LIN {X 0,Y 446.601,Z 250.355,A -85,B 0,C 180,E1 -8646.329,E2 -8646.329} C_VEL
LIN {X 0,Y 446.522,Z 250.36,A -85,B 0,C 180,E1 -8649.06,E2 -8649.06} C_VEL
LIN {X 0,Y 446.522,Z 250.36,A -85,B 0,C 180,E1 -8652.734,E2 -8652.734} C_VEL
LIN {X 0,Y 446.451,Z 250.372,A -85,B 0,C 180,E1 -8656.211,E2 -8656.211} C_VEL
LIN {X 0,Y 446.47,Z 250.369,A -85,B 0,C 180,E1 -8659.307,E2 -8659.307} C_VEL
LIN {X 0,Y 446.419,Z 250.374,A -85,B 0,C 180,E1 -8662.204,E2 -8662.204} C_VEL
LIN {X 0,Y 446.426,Z 250.375,A -85,B 0,C 180,E1 -8665.158,E2 -8665.158} C_VEL
LIN {X 0,Y 446.422,Z 250.373,A -85,B 0,C 180,E1 -8668.187,E2 -8668.187} C_VEL
LIN {X 0,Y 446.415,Z 250.38,A -85,B 0,C 180,E1 -8671.304,E2 -8671.304} C_VEL
LIN {X 0,Y 446.428,Z 250.375,A -85,B 0,C 180,E1 -8674.527,E2 -8674.527} C_VEL
LIN {X 0,Y 446.414,Z 250.379,A -85,B 0,C 180,E1 -8678.08,E2 -8678.08} C_VEL
LIN {X 0,Y 446.421,Z 250.437,A -85,B 0,C 180,E1 -8681.396,E2 -8681.396} C_VEL
LIN {X 0,Y 447.055,Z 254.418,A -85,B 0,C 180,E1 -8685.03,E2 -8685.03} C_VEL
LIN {X 0,Y 447.395,Z 257.531,A -85,B 0,C 180,E1 -8687.592,E2 -8687.592} C_VEL
LIN {X 0,Y 447.38,Z 261.124,A -85,B 0,C 180,E1 -8690.336,E2 -8690.336} C_VEL
LIN {X 0,Y 447.027,Z 265.384,A -85,B 0,C 180,E1 -8693.315,E2 -8693.315} C_VEL
LIN {X 0,Y 446.739,Z 270.172,A -85,B 0,C 180,E1 -8696.494,E2 -8696.494} C_VEL
LIN {X 0,Y 446.406,Z 275.403,A -85,B 0,C 180,E1 -8699.749,E2 -8699.749} C_VEL
LIN {X 0,Y 446.193,Z 280.555,A -85,B 0,C 180,E1 -8702.821,E2 -8702.821} C_VEL
LIN {X 0,Y 445.943,Z 285.793,A -85,B 0,C 180,E1 -8705.811,E2 -8705.811} C_VEL
LIN {X 0,Y 445.831,Z 291.111,A -85,B 0,C 180,E1 -8708.742,E2 -8708.742} C_VEL
LIN {X 0,Y 445.64,Z 296.456,A -85,B 0,C 180,E1 -8711.615,E2 -8711.615} C_VEL
LIN {X 0,Y 445.564,Z 300.748,A -85,B 0,C 180,E1 -8713.868,E2 -8713.868} C_VEL
LIN {X 0,Y 447.507,Z 311.304,A -85,B 0,C 180,E1 -8714.232,E2 -8714.232} C_VEL
LIN {X 0,Y 449.155,Z 321.497,A -85,B 0,C 180,E1 -8714.69,E2 -8714.69} C_VEL
LIN {X 0,Y 449.183,Z 328.569,A -85,B 0,C 180,E1 -8715.039,E2 -8715.039} C_VEL
LIN {X 0,Y 448.687,Z 338.087,A -85,B 0,C 180,E1 -8715.602,E2 -8715.602} C_VEL
LIN {X 0,Y 448.174,Z 347.367,A -85,B 0,C 180,E1 -8716.28,E2 -8716.28} C_VEL
LIN {X 0,Y 447.792,Z 355.767,A -85,B 0,C 180,E1 -8717.021,E2 -8717.021} C_VEL
LIN {X 0,Y 447.286,Z 364.854,A -85,B 0,C 180,E1 -8717.984,E2 -8717.984} C_VEL
LIN {X 0,Y 446.839,Z 372.076,A -85,B 0,C 180,E1 -8718.891,E2 -8718.891} C_VEL
LIN {X 0,Y 446.495,Z 378.281,A -85,B 0,C 180,E1 -8719.801,E2 -8719.801} C_VEL
LIN {X 0,Y 446.129,Z 384.821,A -85,B 0,C 180,E1 -8720.936,E2 -8720.936} C_VEL
LIN {X 0,Y 445.891,Z 389.324,A -85,B 0,C 180,E1 -8721.845,E2 -8721.845} C_VEL
LIN {X 0,Y 445.666,Z 394.973,A -85,B 0,C 180,E1 -8723.253,E2 -8723.253} C_VEL
LIN {X 0,Y 445.537,Z 399.142,A -85,B 0,C 180,E1 -8724.569,E2 -8724.569} C_VEL
LIN {X 0,Y 445.431,Z 401.507,A -85,B 0,C 180,E1 -8725.475,E2 -8725.475} C_VEL
LIN {X 0,Y 445.391,Z 403.304,A -85,B 0,C 180,E1 -8726.381,E2 -8726.381} C_VEL
LIN {X 0,Y 445.357,Z 405.747,A -85,B 0,C 180,E1 -8728.191,E2 -8728.191} C_VEL
LIN {X 0,Y 445.32,Z 406.334,A -85,B 0,C 180,E1 -8729.096,E2 -8729.096} C_VEL
LIN {X 0,Y 445.32,Z 406.334,A -85,B 0,C 180,E1 -8730.904,E2 -8730.904} C_VEL
LIN {X 0,Y 445.357,Z 405.747,A -85,B 0,C 180,E1 -8731.809,E2 -8731.809} C_VEL
LIN {X 0,Y 445.391,Z 403.304,A -85,B 0,C 180,E1 -8733.619,E2 -8733.619} C_VEL
LIN {X 0,Y 445.503,Z 400.359,A -85,B 0,C 180,E1 -8734.977,E2 -8734.977} C_VEL
LIN {X 0,Y 445.59,Z 396.371,A -85,B 0,C 180,E1 -8736.339,E2 -8736.339} C_VEL
LIN {X 0,Y 445.768,Z 391.24,A -85,B 0,C 180,E1 -8737.701,E2 -8737.701} C_VEL
LIN {X 0,Y 446.082,Z 385.978,A -85,B 0,C 180,E1 -8738.836,E2 -8738.836} C_VEL
LIN {X 0,Y 446.427,Z 379.658,A -85,B 0,C 180,E1 -8739.972,E2 -8739.972} C_VEL
LIN {X 0,Y 446.724,Z 373.703,A -85,B 0,C 180,E1 -8740.882,E2 -8740.882} C_VEL
LIN {X 0,Y 447.158,Z 366.773,A -85,B 0,C 180,E1 -8741.79,E2 -8741.79} C_VEL
LIN {X 0,Y 447.622,Z 358.589,A -85,B 0,C 180,E1 -8742.698,E2 -8742.698} C_VEL
LIN {X 0,Y 448.02,Z 350.084,A -85,B 0,C 180,E1 -8743.493,E2 -8743.493} C_VEL
LIN {X 0,Y 448.505,Z 341.352,A -85,B 0,C 180,E1 -8744.172,E2 -8744.172} C_VEL
LIN {X 0,Y 449,Z 331.59,A -85,B 0,C 180,E1 -8744.793,E2 -8744.793} C_VEL
LIN {X 0,Y 449.343,Z 322.793,A -85,B 0,C 180,E1 -8745.245,E2 -8745.245} C_VEL
LIN {X 0,Y 447.629,Z 311.904,A -85,B 0,C 180,E1 -8745.743,E2 -8745.743} C_VEL
LIN {X 0,Y 445.696,Z 301.798,A -85,B 0,C 180,E1 -8746.101,E2 -8746.101} C_VEL
LIN {X 0,Y 445.565,Z 300.694,A -85,B 0,C 180,E1 -8746.16,E2 -8746.16} C_VEL
LIN {X 0,Y 445.696,Z 294.655,A -85,B 0,C 180,E1 -8749.338,E2 -8749.338} C_VEL
LIN {X 0,Y 445.858,Z 289.313,A -85,B 0,C 180,E1 -8752.229,E2 -8752.229} C_VEL
LIN {X 0,Y 446.154,Z 282.386,A -85,B 0,C 180,E1 -8756.113,E2 -8756.113} C_VEL
LIN {X 0,Y 446.347,Z 277.096,A -85,B 0,C 180,E1 -8759.216,E2 -8759.216} C_VEL
LIN {X 0,Y 446.615,Z 271.991,A -85,B 0,C 180,E1 -8762.345,E2 -8762.345} C_VEL
LIN {X 0,Y 446.91,Z 266.987,A -85,B 0,C 180,E1 -8765.58,E2 -8765.58} C_VEL
LIN {X 0,Y 447.299,Z 262.126,A -85,B 0,C 180,E1 -8768.937,E2 -8768.937} C_VEL
LIN {X 0,Y 447.437,Z 258.971,A -85,B 0,C 180,E1 -8771.276,E2 -8771.276} C_VEL
LIN {X 0,Y 447.266,Z 255.884,A -85,B 0,C 180,E1 -8773.739,E2 -8773.739} C_VEL
LIN {X 0,Y 446.779,Z 252.867,A -85,B 0,C 180,E1 -8776.351,E2 -8776.351} C_VEL
LIN {X 0,Y 446.421,Z 250.435,A -85,B 0,C 180,E1 -8778.604,E2 -8778.604} C_VEL
LIN {X 0,Y 446.412,Z 250.379,A -85,B 0,C 180,E1 -8781.92,E2 -8781.92} C_VEL
LIN {X 0,Y 446.428,Z 250.374,A -85,B 0,C 180,E1 -8785.473,E2 -8785.473} C_VEL
LIN {X 0,Y 446.415,Z 250.38,A -85,B 0,C 180,E1 -8788.696,E2 -8788.696} C_VEL
LIN {X 0,Y 446.43,Z 250.372,A -85,B 0,C 180,E1 -8791.833,E2 -8791.833} C_VEL
LIN {X 0,Y 446.426,Z 250.375,A -85,B 0,C 180,E1 -8794.842,E2 -8794.842} C_VEL
LIN {X 0,Y 446.451,Z 250.375,A -85,B 0,C 180,E1 -8798.242,E2 -8798.242} C_VEL
LIN {X 0,Y 446.44,Z 250.372,A -85,B 0,C 180,E1 -8801.644,E2 -8801.644} C_VEL
LIN {X 0,Y 446.459,Z 250.371,A -85,B 0,C 180,E1 -8804.474,E2 -8804.474} C_VEL
LIN {X 0,Y 446.516,Z 250.362,A -85,B 0,C 180,E1 -8807.379,E2 -8807.379} C_VEL
LIN {X 0,Y 446.522,Z 250.36,A -85,B 0,C 180,E1 -8810.94,E2 -8810.94} C_VEL
LIN {X 0,Y 446.601,Z 250.355,A -85,B 0,C 180,E1 -8813.671,E2 -8813.671} C_VEL
LIN {X 0,Y 446.646,Z 250.347,A -85,B 0,C 180,E1 -8817.289,E2 -8817.289} C_VEL
LIN {X 0,Y 446.709,Z 250.341,A -85,B 0,C 180,E1 -8819.995,E2 -8819.995} C_VEL
LIN {X 0,Y 446.669,Z 250.342,A -85,B 0,C 180,E1 -8822.7,E2 -8822.7} C_VEL
LIN {X 0,Y 446.614,Z 250.349,A -85,B 0,C 180,E1 -8826.318,E2 -8826.318} C_VEL
LIN {X 0,Y 446.516,Z 250.364,A -85,B 0,C 180,E1 -8829.05,E2 -8829.05} C_VEL
LIN {X 0,Y 446.504,Z 250.364,A -85,B 0,C 180,E1 -8832.724,E2 -8832.724} C_VEL
LIN {X 0,Y 446.467,Z 250.367,A -85,B 0,C 180,E1 -8836.453,E2 -8836.453} C_VEL
LIN {X 0,Y 446.444,Z 250.375,A -85,B 0,C 180,E1 -8839.298,E2 -8839.298} C_VEL
LIN {X 0,Y 446.391,Z 250.377,A -85,B 0,C 180,E1 -8842.194,E2 -8842.194} C_VEL
LIN {X 0,Y 446.417,Z 250.378,A -85,B 0,C 180,E1 -8845.147,E2 -8845.147} C_VEL
LIN {X 0,Y 446.453,Z 250.369,A -85,B 0,C 180,E1 -8848.173,E2 -8848.173} C_VEL
LIN {X 0,Y 446.383,Z 250.377,A -85,B 0,C 180,E1 -8851.769,E2 -8851.769} C_VEL
LIN {X 0,Y 446.393,Z 250.382,A -85,B 0,C 180,E1 -8854.517,E2 -8854.517} C_VEL
LIN {X 0,Y 446.372,Z 250.381,A -85,B 0,C 180,E1 -8858.073,E2 -8858.073} C_VEL
LIN {X 0,Y 446.393,Z 250.376,A -85,B 0,C 180,E1 -8861.385,E2 -8861.385} C_VEL
LIN {X 0,Y 446.411,Z 250.375,A -85,B 0,C 180,E1 -8864.892,E2 -8864.892} C_VEL
LIN {X 0,Y 446.403,Z 250.376,A -85,B 0,C 180,E1 -8867.715,E2 -8867.715} C_VEL
LIN {X 0,Y 446.423,Z 250.373,A -85,B 0,C 180,E1 -8870.972,E2 -8870.972} C_VEL
LIN {X 0,Y 446.367,Z 250.383,A -85,B 0,C 180,E1 -8874.37,E2 -8874.37} C_VEL
LIN {X 0,Y 446.373,Z 250.382,A -85,B 0,C 180,E1 -8877.635,E2 -8877.635} C_VEL
LIN {X 0,Y 446.411,Z 250.374,A -85,B 0,C 180,E1 -8880.789,E2 -8880.789} C_VEL
LIN {X 0,Y 446.418,Z 250.38,A -85,B 0,C 180,E1 -8883.845,E2 -8883.845} C_VEL
LIN {X 0,Y 446.387,Z 250.377,A -85,B 0,C 180,E1 -8886.821,E2 -8886.821} C_VEL
LIN {X 0,Y 446.397,Z 250.382,A -85,B 0,C 180,E1 -8889.735,E2 -8889.735} C_VEL
LIN {X 0,Y 446.408,Z 250.378,A -85,B 0,C 180,E1 -8892.595,E2 -8892.595} C_VEL
LIN {X 0,Y 446.423,Z 250.38,A -85,B 0,C 180,E1 -8895.411,E2 -8895.411} C_VEL
LIN {X 0,Y 446.482,Z 250.368,A -85,B 0,C 180,E1 -8898.192,E2 -8898.192} C_VEL
LIN {X 0,Y 446.54,Z 250.362,A -85,B 0,C 180,E1 -8901.857,E2 -8901.857} C_VEL
LIN {X 0,Y 446.591,Z 250.356,A -85,B 0,C 180,E1 -8904.582,E2 -8904.582} C_VEL
LIN {X 0,Y 446.56,Z 250.36,A -85,B 0,C 180,E1 -8906.966,E2 -8906.966} C_VEL
LIN {X 0,Y 446.041,Z 250.428,A -85,B 0,C 180,E1 -8907.719,E2 -8907.719} C_VEL
LIN {X 0,Y 443.252,Z 250.781,A -85,B 0,C 180,E1 -8908.943,E2 -8908.943} C_VEL
LIN {X 0,Y 440.785,Z 251.087,A -85,B 0,C 180,E1 -8909.93,E2 -8909.93} C_VEL
LIN {X 0,Y 439.691,Z 251.219,A -85,B 0,C 180,E1 -8910.693,E2 -8910.693} C_VEL
LIN {X 0,Y 439.588,Z 251.229,A -85,B 0,C 180,E1 -8910.952,E2 -8910.952} C_VEL
LIN {X 0,Y 439.599,Z 251.229,A -85,B 0,C 180,E1 -8912.749,E2 -8912.749} C_VEL
LIN {X 0,Y 439.567,Z 251.233,A -85,B 0,C 180,E1 -8916.426,E2 -8916.426} C_VEL
LIN {X 0,Y 439.452,Z 251.246,A -85,B 0,C 180,E1 -8919.202,E2 -8919.202} C_VEL
LIN {X 0,Y 439.44,Z 251.25,A -85,B 0,C 180,E1 -8922.728,E2 -8922.728} C_VEL
LIN {X 0,Y 439.397,Z 251.254,A -85,B 0,C 180,E1 -8926.357,E2 -8926.357} C_VEL
LIN {X 0,Y 439.373,Z 251.251,A -85,B 0,C 180,E1 -8929.627,E2 -8929.627} C_VEL
LIN {X 0,Y 439.325,Z 251.261,A -85,B 0,C 180,E1 -8932.577,E2 -8932.577} C_VEL
LIN {X 0,Y 439.355,Z 251.254,A -85,B 0,C 180,E1 -8935.587,E2 -8935.587} C_VEL
LIN {X 0,Y 439.367,Z 251.253,A -85,B 0,C 180,E1 -8938.676,E2 -8938.676} C_VEL
LIN {X 0,Y 439.328,Z 251.264,A -85,B 0,C 180,E1 -8942.037,E2 -8942.037} C_VEL
LIN {X 0,Y 439.341,Z 251.256,A -85,B 0,C 180,E1 -8945.345,E2 -8945.345} C_VEL
LIN {X 0,Y 439.347,Z 251.254,A -85,B 0,C 180,E1 -8948.598,E2 -8948.598} C_VEL
LIN {X 0,Y 439.355,Z 251.255,A -85,B 0,C 180,E1 -8951.264,E2 -8951.264} C_VEL
LIN {X 0,Y 439.363,Z 251.252,A -85,B 0,C 180,E1 -8954.733,E2 -8954.733} C_VEL
LIN {X 0,Y 439.367,Z 251.256,A -85,B 0,C 180,E1 -8957.803,E2 -8957.803} C_VEL
LIN {X 0,Y 439.347,Z 251.254,A -85,B 0,C 180,E1 -8960.229,E2 -8960.229} C_VEL
LIN {X 0,Y 439.336,Z 251.259,A -85,B 0,C 180,E1 -8963.718,E2 -8963.718} C_VEL
LIN {X 0,Y 439.337,Z 251.26,A -85,B 0,C 180,E1 -8967.06,E2 -8967.06} C_VEL
LIN {X 0,Y 439.348,Z 251.254,A -85,B 0,C 180,E1 -8970.28,E2 -8970.28} C_VEL
LIN {X 0,Y 439.398,Z 251.251,A -85,B 0,C 180,E1 -8973.402,E2 -8973.402} C_VEL
LIN {X 0,Y 439.357,Z 251.254,A -85,B 0,C 180,E1 -8976.435,E2 -8976.435} C_VEL
LIN {X 0,Y 439.362,Z 251.254,A -85,B 0,C 180,E1 -8979.403,E2 -8979.403} C_VEL
LIN {X 0,Y 439.381,Z 251.251,A -85,B 0,C 180,E1 -8982.314,E2 -8982.314} C_VEL
LIN {X 0,Y 439.423,Z 251.247,A -85,B 0,C 180,E1 -8985.18,E2 -8985.18} C_VEL
LIN {X 0,Y 439.466,Z 251.24,A -85,B 0,C 180,E1 -8988.007,E2 -8988.007} C_VEL
LIN {X 0,Y 439.489,Z 251.236,A -85,B 0,C 180,E1 -8991.731,E2 -8991.731} C_VEL
LIN {X 0,Y 439.596,Z 251.23,A -85,B 0,C 180,E1 -8994.501,E2 -8994.501} C_VEL
LIN {X 0,Y 439.623,Z 251.225,A -85,B 0,C 180,E1 -8998.173,E2 -8998.173} C_VEL
LIN {X 0,Y 439.577,Z 251.226,A -85,B 0,C 180,E1 -9000.921,E2 -9000.921} C_VEL
LIN {X 0,Y 439.597,Z 251.224,A -85,B 0,C 180,E1 -9002.754,E2 -9002.754} C_VEL
LIN {X 0,Y 439.554,Z 251.232,A -85,B 0,C 180,E1 -9006.431,E2 -9006.431} C_VEL
LIN {X 0,Y 439.487,Z 251.237,A -85,B 0,C 180,E1 -9009.207,E2 -9009.207} C_VEL
LIN {X 0,Y 439.465,Z 251.239,A -85,B 0,C 180,E1 -9012.942,E2 -9012.942} C_VEL
LIN {X 0,Y 439.398,Z 251.249,A -85,B 0,C 180,E1 -9016.33,E2 -9016.33} C_VEL
LIN {X 0,Y 439.403,Z 251.253,A -85,B 0,C 180,E1 -9019.631,E2 -9019.631} C_VEL
LIN {X 0,Y 439.365,Z 251.252,A -85,B 0,C 180,E1 -9022.58,E2 -9022.58} C_VEL
LIN {X 0,Y 439.372,Z 251.258,A -85,B 0,C 180,E1 -9025.591,E2 -9025.591} C_VEL
LIN {X 0,Y 439.388,Z 251.249,A -85,B 0,C 180,E1 -9028.68,E2 -9028.68} C_VEL
LIN {X 0,Y 439.369,Z 251.252,A -85,B 0,C 180,E1 -9032.032,E2 -9032.032} C_VEL
LIN {X 0,Y 439.397,Z 251.255,A -85,B 0,C 180,E1 -9035.342,E2 -9035.342} C_VEL
LIN {X 0,Y 439.367,Z 251.258,A -85,B 0,C 180,E1 -9038.601,E2 -9038.601} C_VEL
LIN {X 0,Y 439.366,Z 251.259,A -85,B 0,C 180,E1 -9040.986,E2 -9040.986} C_VEL
LIN {X 0,Y 439.857,Z 254.468,A -85,B 0,C 180,E1 -9044.029,E2 -9044.029} C_VEL
LIN {X 0,Y 440.258,Z 257.496,A -85,B 0,C 180,E1 -9046.653,E2 -9046.653} C_VEL
LIN {X 0,Y 440.412,Z 260.61,A -85,B 0,C 180,E1 -9049.137,E2 -9049.137} C_VEL
LIN {X 0,Y 440.247,Z 263.779,A -85,B 0,C 180,E1 -9051.496,E2 -9051.496} C_VEL
LIN {X 0,Y 439.853,Z 268.663,A -85,B 0,C 180,E1 -9054.886,E2 -9054.886} C_VEL
LIN {X 0,Y 439.518,Z 273.66,A -85,B 0,C 180,E1 -9058.152,E2 -9058.152} C_VEL
LIN {X 0,Y 439.229,Z 279.316,A -85,B 0,C 180,E1 -9061.652,E2 -9061.652} C_VEL
LIN {X 0,Y 438.998,Z 283.948,A -85,B 0,C 180,E1 -9064.39,E2 -9064.39} C_VEL
LIN {X 0,Y 438.785,Z 289.194,A -85,B 0,C 180,E1 -9067.394,E2 -9067.394} C_VEL
LIN {X 0,Y 438.622,Z 294.503,A -85,B 0,C 180,E1 -9070.338,E2 -9070.338} C_VEL
LIN {X 0,Y 438.492,Z 300.563,A -85,B 0,C 180,E1 -9073.6,E2 -9073.6} C_VEL
LIN {X 0,Y 440.394,Z 310.801,A -85,B 0,C 180,E1 -9073.961,E2 -9073.961} C_VEL
LIN {X 0,Y 442.113,Z 321.28,A -85,B 0,C 180,E1 -9074.44,E2 -9074.44} C_VEL
LIN {X 0,Y 442.419,Z 326.322,A -85,B 0,C 180,E1 -9074.687,E2 -9074.687} C_VEL
LIN {X 0,Y 441.788,Z 337.875,A -85,B 0,C 180,E1 -9075.372,E2 -9075.372} C_VEL
LIN {X 0,Y 441.254,Z 347.155,A -85,B 0,C 180,E1 -9076.061,E2 -9076.061} C_VEL
LIN {X 0,Y 440.8,Z 356.338,A -85,B 0,C 180,E1 -9076.892,E2 -9076.892} C_VEL
LIN {X 0,Y 440.322,Z 364.642,A -85,B 0,C 180,E1 -9077.791,E2 -9077.791} C_VEL
LIN {X 0,Y 439.837,Z 371.864,A -85,B 0,C 180,E1 -9078.712,E2 -9078.712} C_VEL
LIN {X 0,Y 439.478,Z 378.069,A -85,B 0,C 180,E1 -9079.636,E2 -9079.636} C_VEL
LIN {X 0,Y 439.082,Z 384.609,A -85,B 0,C 180,E1 -9080.79,E2 -9080.79} C_VEL
LIN {X 0,Y 438.838,Z 389.112,A -85,B 0,C 180,E1 -9081.713,E2 -9081.713} C_VEL
LIN {X 0,Y 438.601,Z 394.606,A -85,B 0,C 180,E1 -9083.098,E2 -9083.098} C_VEL
LIN {X 0,Y 438.438,Z 398.93,A -85,B 0,C 180,E1 -9084.481,E2 -9084.481} C_VEL
LIN {X 0,Y 438.361,Z 401.296,A -85,B 0,C 180,E1 -9085.402,E2 -9085.402} C_VEL
LIN {X 0,Y 438.337,Z 404.481,A -85,B 0,C 180,E1 -9087.243,E2 -9087.243} C_VEL
LIN {X 0,Y 438.28,Z 405.537,A -85,B 0,C 180,E1 -9088.162,E2 -9088.162} C_VEL
LIN {X 0,Y 438.235,Z 406.123,A -85,B 0,C 180,E1 -9089.081,E2 -9089.081} C_VEL
LIN {X 0,Y 438.235,Z 406.123,A -85,B 0,C 180,E1 -9090.919,E2 -9090.919} C_VEL
LIN {X 0,Y 438.28,Z 405.537,A -85,B 0,C 180,E1 -9091.838,E2 -9091.838} C_VEL
LIN {X 0,Y 438.293,Z 403.093,A -85,B 0,C 180,E1 -9093.677,E2 -9093.677} C_VEL
LIN {X 0,Y 438.416,Z 400.147,A -85,B 0,C 180,E1 -9095.058,E2 -9095.058} C_VEL
LIN {X 0,Y 438.518,Z 396.159,A -85,B 0,C 180,E1 -9096.441,E2 -9096.441} C_VEL
LIN {X 0,Y 438.725,Z 391.028,A -85,B 0,C 180,E1 -9097.826,E2 -9097.826} C_VEL
LIN {X 0,Y 439.041,Z 385.766,A -85,B 0,C 180,E1 -9098.979,E2 -9098.979} C_VEL
LIN {X 0,Y 439.401,Z 379.446,A -85,B 0,C 180,E1 -9100.133,E2 -9100.133} C_VEL
LIN {X 0,Y 439.711,Z 373.491,A -85,B 0,C 180,E1 -9101.058,E2 -9101.058} C_VEL
LIN {X 0,Y 440.185,Z 366.561,A -85,B 0,C 180,E1 -9101.979,E2 -9101.979} C_VEL
LIN {X 0,Y 440.663,Z 358.377,A -85,B 0,C 180,E1 -9102.902,E2 -9102.902} C_VEL
LIN {X 0,Y 441.076,Z 350.155,A -85,B 0,C 180,E1 -9103.684,E2 -9103.684} C_VEL
LIN {X 0,Y 441.596,Z 341.14,A -85,B 0,C 180,E1 -9104.399,E2 -9104.399} C_VEL
LIN {X 0,Y 442.143,Z 331.379,A -85,B 0,C 180,E1 -9105.028,E2 -9105.028} C_VEL
LIN {X 0,Y 442.473,Z 323.87,A -85,B 0,C 180,E1 -9105.429,E2 -9105.429} C_VEL
LIN {X 0,Y 440.716,Z 312.516,A -85,B 0,C 180,E1 -9105.969,E2 -9105.969} C_VEL
LIN {X 0,Y 438.599,Z 301.625,A -85,B 0,C 180,E1 -9106.368,E2 -9106.368} C_VEL
LIN {X 0,Y 438.492,Z 300.563,A -85,B 0,C 180,E1 -9106.4,E2 -9106.4} C_VEL
LIN {X 0,Y 438.62,Z 294.5,A -85,B 0,C 180,E1 -9109.662,E2 -9109.662} C_VEL
LIN {X 0,Y 438.786,Z 289.188,A -85,B 0,C 180,E1 -9112.606,E2 -9112.606} C_VEL
LIN {X 0,Y 439.091,Z 282.717,A -85,B 0,C 180,E1 -9116.316,E2 -9116.316} C_VEL
LIN {X 0,Y 439.247,Z 278.751,A -85,B 0,C 180,E1 -9118.685,E2 -9118.685} C_VEL
LIN {X 0,Y 439.537,Z 273.324,A -85,B 0,C 180,E1 -9122.061,E2 -9122.061} C_VEL
LIN {X 0,Y 439.854,Z 268.655,A -85,B 0,C 180,E1 -9125.113,E2 -9125.113} C_VEL
LIN {X 0,Y 440.257,Z 263.739,A -85,B 0,C 180,E1 -9128.533,E2 -9128.533} C_VEL
LIN {X 0,Y 440.421,Z 259.902,A -85,B 0,C 180,E1 -9131.406,E2 -9131.406} C_VEL
LIN {X 0,Y 440.209,Z 256.623,A -85,B 0,C 180,E1 -9134.071,E2 -9134.071} C_VEL
LIN {X 0,Y 439.636,Z 253.006,A -85,B 0,C 180,E1 -9137.336,E2 -9137.336} C_VEL
LIN {X 0,Y 439.366,Z 251.259,A -85,B 0,C 180,E1 -9139.014,E2 -9139.014} C_VEL
LIN {X 0,Y 439.349,Z 251.26,A -85,B 0,C 180,E1 -9142.561,E2 -9142.561} C_VEL
LIN {X 0,Y 439.401,Z 251.254,A -85,B 0,C 180,E1 -9144.84,E2 -9144.84} C_VEL
LIN {X 0,Y 439.373,Z 251.253,A -85,B 0,C 180,E1 -9148.135,E2 -9148.135} C_VEL
LIN {X 0,Y 439.393,Z 251.248,A -85,B 0,C 180,E1 -9151.606,E2 -9151.606} C_VEL
LIN {X 0,Y 439.372,Z 251.258,A -85,B 0,C 180,E1 -9154.409,E2 -9154.409} C_VEL
LIN {X 0,Y 439.365,Z 251.252,A -85,B 0,C 180,E1 -9157.42,E2 -9157.42} C_VEL
LIN {X 0,Y 439.444,Z 251.245,A -85,B 0,C 180,E1 -9160.659,E2 -9160.659} C_VEL
LIN {X 0,Y 439.418,Z 251.252,A -85,B 0,C 180,E1 -9164.218,E2 -9164.218} C_VEL
LIN {X 0,Y 439.485,Z 251.237,A -85,B 0,C 180,E1 -9167.281,E2 -9167.281} C_VEL
LIN {X 0,Y 439.487,Z 251.237,A -85,B 0,C 180,E1 -9170.793,E2 -9170.793} C_VEL
LIN {X 0,Y 439.554,Z 251.232,A -85,B 0,C 180,E1 -9173.569,E2 -9173.569} C_VEL
LIN {X 0,Y 439.4,Z 251.25,A -85,B 0,C 180,E1 -9175.408,E2 -9175.408} C_VEL
LIN {X 0,Y 439.618,Z 251.223,A -85,B 0,C 180,E1 -9178.163,E2 -9178.163} C_VEL
LIN {X 0,Y 439.66,Z 251.219,A -85,B 0,C 180,E1 -9179.995,E2 -9179.995} C_VEL
LIN {X 0,Y 439.619,Z 251.22,A -85,B 0,C 180,E1 -9182.743,E2 -9182.743} C_VEL
LIN {X 0,Y 439.585,Z 251.224,A -85,B 0,C 180,E1 -9186.42,E2 -9186.42} C_VEL
LIN {X 0,Y 439.479,Z 251.242,A -85,B 0,C 180,E1 -9189.196,E2 -9189.196} C_VEL
LIN {X 0,Y 439.447,Z 251.245,A -85,B 0,C 180,E1 -9192.932,E2 -9192.932} C_VEL
LIN {X 0,Y 439.425,Z 251.244,A -85,B 0,C 180,E1 -9196.342,E2 -9196.342} C_VEL
LIN {X 0,Y 439.378,Z 251.252,A -85,B 0,C 180,E1 -9199.62,E2 -9199.62} C_VEL
LIN {X 0,Y 439.337,Z 251.257,A -85,B 0,C 180,E1 -9202.57,E2 -9202.57} C_VEL
LIN {X 0,Y 439.37,Z 251.252,A -85,B 0,C 180,E1 -9205.579,E2 -9205.579} C_VEL
LIN {X 0,Y 439.385,Z 251.255,A -85,B 0,C 180,E1 -9208.668,E2 -9208.668} C_VEL
LIN {X 0,Y 439.334,Z 251.256,A -85,B 0,C 180,E1 -9212.024,E2 -9212.024} C_VEL
LIN {X 0,Y 439.358,Z 251.253,A -85,B 0,C 180,E1 -9215.335,E2 -9215.335} C_VEL
LIN {X 0,Y 439.329,Z 251.263,A -85,B 0,C 180,E1 -9218.591,E2 -9218.591} C_VEL
LIN {X 0,Y 439.351,Z 251.254,A -85,B 0,C 180,E1 -9221.252,E2 -9221.252} C_VEL
LIN {X 0,Y 439.363,Z 251.255,A -85,B 0,C 180,E1 -9224.723,E2 -9224.723} C_VEL
LIN {X 0,Y 439.363,Z 251.254,A -85,B 0,C 180,E1 -9227.793,E2 -9227.793} C_VEL
LIN {X 0,Y 439.401,Z 251.254,A -85,B 0,C 180,E1 -9230.225,E2 -9230.225} C_VEL
LIN {X 0,Y 439.323,Z 251.26,A -85,B 0,C 180,E1 -9233.709,E2 -9233.709} C_VEL
LIN {X 0,Y 439.32,Z 251.257,A -85,B 0,C 180,E1 -9237.05,E2 -9237.05} C_VEL
LIN {X 0,Y 439.339,Z 251.258,A -85,B 0,C 180,E1 -9240.272,E2 -9240.272} C_VEL
LIN {X 0,Y 439.374,Z 251.255,A -85,B 0,C 180,E1 -9243.585,E2 -9243.585} C_VEL
LIN {X 0,Y 439.339,Z 251.255,A -85,B 0,C 180,E1 -9246.427,E2 -9246.427} C_VEL
LIN {X 0,Y 439.351,Z 251.258,A -85,B 0,C 180,E1 -9249.396,E2 -9249.396} C_VEL
LIN {X 0,Y 439.375,Z 251.254,A -85,B 0,C 180,E1 -9252.308,E2 -9252.308} C_VEL
LIN {X 0,Y 439.4,Z 251.254,A -85,B 0,C 180,E1 -9255.173,E2 -9255.173} C_VEL
LIN {X 0,Y 439.448,Z 251.244,A -85,B 0,C 180,E1 -9258.001,E2 -9258.001} C_VEL
LIN {X 0,Y 439.488,Z 251.241,A -85,B 0,C 180,E1 -9261.725,E2 -9261.725} C_VEL
LIN {X 0,Y 439.566,Z 251.23,A -85,B 0,C 180,E1 -9264.495,E2 -9264.495} C_VEL
LIN {X 0,Y 439.571,Z 251.229,A -85,B 0,C 180,E1 -9268.168,E2 -9268.168} C_VEL
LIN {X 0,Y 439.697,Z 251.215,A -85,B 0,C 180,E1 -9270,E2 -9270} C_VEL
LIN {X 0,Y 439.588,Z 251.229,A -85,B 0,C 180,E1 -9270.952,E2 -9270.952} C_VEL
LIN {X 0,Y 438.85,Z 251.319,A -85,B 0,C 180,E1 -9271.716,E2 -9271.716} C_VEL
LIN {X 0,Y 435.861,Z 251.694,A -85,B 0,C 180,E1 -9272.955,E2 -9272.955} C_VEL
LIN {X 0,Y 433.412,Z 251.999,A -85,B 0,C 180,E1 -9273.955,E2 -9273.955} C_VEL
LIN {X 0,Y 432.44,Z 252.12,A -85,B 0,C 180,E1 -9274.73,E2 -9274.73} C_VEL
LIN {X 0,Y 432.402,Z 252.122,A -85,B 0,C 180,E1 -9274.992,E2 -9274.992} C_VEL
LIN {X 0,Y 432.52,Z 252.109,A -85,B 0,C 180,E1 -9277.68,E2 -9277.68} C_VEL
LIN {X 0,Y 432.35,Z 252.13,A -85,B 0,C 180,E1 -9281.248,E2 -9281.248} C_VEL
LIN {X 0,Y 432.329,Z 252.133,A -85,B 0,C 180,E1 -9284.113,E2 -9284.113} C_VEL
LIN {X 0,Y 432.338,Z 252.132,A -85,B 0,C 180,E1 -9287.014,E2 -9287.014} C_VEL
LIN {X 0,Y 432.32,Z 252.132,A -85,B 0,C 180,E1 -9289.961,E2 -9289.961} C_VEL
LIN {X 0,Y 432.274,Z 252.136,A -85,B 0,C 180,E1 -9292.966,E2 -9292.966} C_VEL
LIN {X 0,Y 432.31,Z 252.136,A -85,B 0,C 180,E1 -9296.035,E2 -9296.035} C_VEL
LIN {X 0,Y 432.295,Z 252.132,A -85,B 0,C 180,E1 -9299.19,E2 -9299.19} C_VEL
LIN {X 0,Y 432.277,Z 252.139,A -85,B 0,C 180,E1 -9302.299,E2 -9302.299} C_VEL
LIN {X 0,Y 432.286,Z 252.134,A -85,B 0,C 180,E1 -9304.681,E2 -9304.681} C_VEL
LIN {X 0,Y 432.301,Z 252.135,A -85,B 0,C 180,E1 -9308.153,E2 -9308.153} C_VEL
LIN {X 0,Y 432.324,Z 252.134,A -85,B 0,C 180,E1 -9311.613,E2 -9311.613} C_VEL
LIN {X 0,Y 432.332,Z 252.129,A -85,B 0,C 180,E1 -9314.346,E2 -9314.346} C_VEL
LIN {X 0,Y 432.321,Z 252.13,A -85,B 0,C 180,E1 -9317.014,E2 -9317.014} C_VEL
LIN {X 0,Y 432.292,Z 252.136,A -85,B 0,C 180,E1 -9319.826,E2 -9319.826} C_VEL
LIN {X 0,Y 432.267,Z 252.139,A -85,B 0,C 180,E1 -9323.027,E2 -9323.027} C_VEL
LIN {X 0,Y 432.323,Z 252.13,A -85,B 0,C 180,E1 -9326.002,E2 -9326.002} C_VEL
LIN {X 0,Y 432.313,Z 252.134,A -85,B 0,C 180,E1 -9329.496,E2 -9329.496} C_VEL
LIN {X 0,Y 432.36,Z 252.129,A -85,B 0,C 180,E1 -9332.934,E2 -9332.934} C_VEL
LIN {X 0,Y 432.341,Z 252.127,A -85,B 0,C 180,E1 -9336.029,E2 -9336.029} C_VEL
LIN {X 0,Y 432.324,Z 252.135,A -85,B 0,C 180,E1 -9339.052,E2 -9339.052} C_VEL
LIN {X 0,Y 432.337,Z 252.127,A -85,B 0,C 180,E1 -9342.016,E2 -9342.016} C_VEL
LIN {X 0,Y 432.371,Z 252.128,A -85,B 0,C 180,E1 -9344.932,E2 -9344.932} C_VEL
LIN {X 0,Y 432.441,Z 252.114,A -85,B 0,C 180,E1 -9347.809,E2 -9347.809} C_VEL
LIN {X 0,Y 432.449,Z 252.113,A -85,B 0,C 180,E1 -9351.595,E2 -9351.595} C_VEL
LIN {X 0,Y 432.572,Z 252.104,A -85,B 0,C 180,E1 -9354.412,E2 -9354.412} C_VEL
LIN {X 0,Y 432.592,Z 252.1,A -85,B 0,C 180,E1 -9358.144,E2 -9358.144} C_VEL
LIN {X 0,Y 432.538,Z 252.103,A -85,B 0,C 180,E1 -9360.936,E2 -9360.936} C_VEL
LIN {X 0,Y 432.551,Z 252.102,A -85,B 0,C 180,E1 -9362.799,E2 -9362.799} C_VEL
LIN {X 0,Y 432.511,Z 252.108,A -85,B 0,C 180,E1 -9366.536,E2 -9366.536} C_VEL
LIN {X 0,Y 432.432,Z 252.116,A -85,B 0,C 180,E1 -9369.358,E2 -9369.358} C_VEL
LIN {X 0,Y 432.431,Z 252.115,A -85,B 0,C 180,E1 -9372.808,E2 -9372.808} C_VEL
LIN {X 0,Y 432.358,Z 252.126,A -85,B 0,C 180,E1 -9376.457,E2 -9376.457} C_VEL
LIN {X 0,Y 432.389,Z 252.125,A -85,B 0,C 180,E1 -9379.489,E2 -9379.489} C_VEL
LIN {X 0,Y 432.314,Z 252.131,A -85,B 0,C 180,E1 -9382.969,E2 -9382.969} C_VEL
LIN {X 0,Y 432.323,Z 252.131,A -85,B 0,C 180,E1 -9386.039,E2 -9386.039} C_VEL
LIN {X 0,Y 432.329,Z 252.132,A -85,B 0,C 180,E1 -9389.193,E2 -9389.193} C_VEL
LIN {X 0,Y 432.327,Z 252.128,A -85,B 0,C 180,E1 -9392.447,E2 -9392.447} C_VEL
LIN {X 0,Y 432.343,Z 252.131,A -85,B 0,C 180,E1 -9395.821,E2 -9395.821} C_VEL
LIN {X 0,Y 432.31,Z 252.138,A -85,B 0,C 180,E1 -9399.351,E2 -9399.351} C_VEL
LIN {X 0,Y 432.3,Z 252.138,A -85,B 0,C 180,E1 -9400.568,E2 -9400.568} C_VEL
LIN {X 0,Y 432.706,Z 254.575,A -85,B 0,C 180,E1 -9403.04,E2 -9403.04} C_VEL
LIN {X 0,Y 433.161,Z 257.588,A -85,B 0,C 180,E1 -9405.761,E2 -9405.761} C_VEL
LIN {X 0,Y 433.401,Z 260.674,A -85,B 0,C 180,E1 -9408.33,E2 -9408.33} C_VEL
LIN {X 0,Y 433.252,Z 264.326,A -85,B 0,C 180,E1 -9411.14,E2 -9411.14} C_VEL
LIN {X 0,Y 432.853,Z 268.726,A -85,B 0,C 180,E1 -9414.279,E2 -9414.279} C_VEL
LIN {X 0,Y 432.639,Z 271.983,A -85,B 0,C 180,E1 -9416.475,E2 -9416.475} C_VEL
LIN {X 0,Y 432.303,Z 276.994,A -85,B 0,C 180,E1 -9419.738,E2 -9419.738} C_VEL
LIN {X 0,Y 432.052,Z 282.128,A -85,B 0,C 180,E1 -9422.906,E2 -9422.906} C_VEL
LIN {X 0,Y 431.792,Z 287.324,A -85,B 0,C 180,E1 -9425.99,E2 -9425.99} C_VEL
LIN {X 0,Y 431.632,Z 292.583,A -85,B 0,C 180,E1 -9429.01,E2 -9429.01} C_VEL
LIN {X 0,Y 431.437,Z 297.899,A -85,B 0,C 180,E1 -9431.971,E2 -9431.971} C_VEL
LIN {X 0,Y 431.409,Z 300.389,A -85,B 0,C 180,E1 -9433.328,E2 -9433.328} C_VEL
LIN {X 0,Y 433.27,Z 310.297,A -85,B 0,C 180,E1 -9433.68,E2 -9433.68} C_VEL
LIN {X 0,Y 434.888,Z 319.767,A -85,B 0,C 180,E1 -9434.115,E2 -9434.115} C_VEL
LIN {X 0,Y 435.558,Z 326.11,A -85,B 0,C 180,E1 -9434.44,E2 -9434.44} C_VEL
LIN {X 0,Y 434.899,Z 337.663,A -85,B 0,C 180,E1 -9435.135,E2 -9435.135} C_VEL
LIN {X 0,Y 434.352,Z 346.943,A -85,B 0,C 180,E1 -9435.834,E2 -9435.834} C_VEL
LIN {X 0,Y 433.933,Z 354.889,A -85,B 0,C 180,E1 -9436.551,E2 -9436.551} C_VEL
LIN {X 0,Y 433.505,Z 362.51,A -85,B 0,C 180,E1 -9437.358,E2 -9437.358} C_VEL
LIN {X 0,Y 432.853,Z 371.651,A -85,B 0,C 180,E1 -9438.528,E2 -9438.528} C_VEL
LIN {X 0,Y 432.469,Z 377.857,A -85,B 0,C 180,E1 -9439.466,E2 -9439.466} C_VEL
LIN {X 0,Y 432.057,Z 384.397,A -85,B 0,C 180,E1 -9440.639,E2 -9440.639} C_VEL
LIN {X 0,Y 431.797,Z 388.9,A -85,B 0,C 180,E1 -9441.577,E2 -9441.577} C_VEL
LIN {X 0,Y 431.532,Z 394.394,A -85,B 0,C 180,E1 -9442.984,E2 -9442.984} C_VEL
LIN {X 0,Y 431.343,Z 398.718,A -85,B 0,C 180,E1 -9444.39,E2 -9444.39} C_VEL
LIN {X 0,Y 431.292,Z 401.085,A -85,B 0,C 180,E1 -9445.327,E2 -9445.327} C_VEL
LIN {X 0,Y 431.234,Z 404.269,A -85,B 0,C 180,E1 -9447.198,E2 -9447.198} C_VEL
LIN {X 0,Y 431.205,Z 405.326,A -85,B 0,C 180,E1 -9448.132,E2 -9448.132} C_VEL
LIN {X 0,Y 431.154,Z 405.913,A -85,B 0,C 180,E1 -9449.066,E2 -9449.066} C_VEL
LIN {X 0,Y 431.154,Z 405.913,A -85,B 0,C 180,E1 -9450.934,E2 -9450.934} C_VEL
LIN {X 0,Y 431.205,Z 405.326,A -85,B 0,C 180,E1 -9451.868,E2 -9451.868} C_VEL
LIN {X 0,Y 431.2,Z 402.881,A -85,B 0,C 180,E1 -9453.738,E2 -9453.738} C_VEL
LIN {X 0,Y 431.331,Z 399.935,A -85,B 0,C 180,E1 -9455.141,E2 -9455.141} C_VEL
LIN {X 0,Y 431.454,Z 395.947,A -85,B 0,C 180,E1 -9456.547,E2 -9456.547} C_VEL
LIN {X 0,Y 431.653,Z 390.816,A -85,B 0,C 180,E1 -9457.955,E2 -9457.955} C_VEL
LIN {X 0,Y 431.974,Z 385.553,A -85,B 0,C 180,E1 -9459.127,E2 -9459.127} C_VEL
LIN {X 0,Y 432.362,Z 379.233,A -85,B 0,C 180,E1 -9460.3,E2 -9460.3} C_VEL
LIN {X 0,Y 432.712,Z 373.278,A -85,B 0,C 180,E1 -9461.239,E2 -9461.239} C_VEL
LIN {X 0,Y 433.226,Z 366.35,A -85,B 0,C 180,E1 -9462.174,E2 -9462.174} C_VEL
LIN {X 0,Y 433.71,Z 358.165,A -85,B 0,C 180,E1 -9463.112,E2 -9463.112} C_VEL
LIN {X 0,Y 434.194,Z 349.328,A -85,B 0,C 180,E1 -9463.96,E2 -9463.96} C_VEL
LIN {X 0,Y 434.721,Z 340.928,A -85,B 0,C 180,E1 -9464.631,E2 -9464.631} C_VEL
LIN {X 0,Y 435.283,Z 331.168,A -85,B 0,C 180,E1 -9465.27,E2 -9465.27} C_VEL
LIN {X 0,Y 435.611,Z 324.946,A -85,B 0,C 180,E1 -9465.618,E2 -9465.618} C_VEL
LIN {X 0,Y 433.7,Z 312.537,A -85,B 0,C 180,E1 -9466.226,E2 -9466.226} C_VEL
LIN {X 0,Y 431.641,Z 301.99,A -85,B 0,C 180,E1 -9466.626,E2 -9466.626} C_VEL
LIN {X 0,Y 431.405,Z 300.355,A -85,B 0,C 180,E1 -9466.69,E2 -9466.69} C_VEL
LIN {X 0,Y 431.545,Z 294.344,A -85,B 0,C 180,E1 -9469.998,E2 -9469.998} C_VEL
LIN {X 0,Y 431.728,Z 289.067,A -85,B 0,C 180,E1 -9472.997,E2 -9472.997} C_VEL
LIN {X 0,Y 432.025,Z 283.052,A -85,B 0,C 180,E1 -9476.523,E2 -9476.523} C_VEL
LIN {X 0,Y 432.212,Z 278.686,A -85,B 0,C 180,E1 -9479.197,E2 -9479.197} C_VEL
LIN {X 0,Y 432.522,Z 273.623,A -85,B 0,C 180,E1 -9482.426,E2 -9482.426} C_VEL
LIN {X 0,Y 432.882,Z 268.656,A -85,B 0,C 180,E1 -9485.765,E2 -9485.765} C_VEL
LIN {X 0,Y 433.274,Z 263.811,A -85,B 0,C 180,E1 -9489.242,E2 -9489.242} C_VEL
LIN {X 0,Y 433.397,Z 260.566,A -85,B 0,C 180,E1 -9491.756,E2 -9491.756} C_VEL
LIN {X 0,Y 433.159,Z 257.352,A -85,B 0,C 180,E1 -9494.443,E2 -9494.443} C_VEL
LIN {X 0,Y 432.683,Z 254.559,A -85,B 0,C 180,E1 -9496.98,E2 -9496.98} C_VEL
LIN {X 0,Y 432.3,Z 252.137,A -85,B 0,C 180,E1 -9499.432,E2 -9499.432} C_VEL
LIN {X 0,Y 432.333,Z 252.133,A -85,B 0,C 180,E1 -9501.846,E2 -9501.846} C_VEL
LIN {X 0,Y 432.334,Z 252.133,A -85,B 0,C 180,E1 -9505.318,E2 -9505.318} C_VEL
LIN {X 0,Y 432.322,Z 252.136,A -85,B 0,C 180,E1 -9508.65,E2 -9508.65} C_VEL
LIN {X 0,Y 432.325,Z 252.129,A -85,B 0,C 180,E1 -9511.868,E2 -9511.868} C_VEL
LIN {X 0,Y 432.327,Z 252.13,A -85,B 0,C 180,E1 -9514.993,E2 -9514.993} C_VEL
LIN {X 0,Y 432.359,Z 252.128,A -85,B 0,C 180,E1 -9518.041,E2 -9518.041} C_VEL
LIN {X 0,Y 432.383,Z 252.122,A -85,B 0,C 180,E1 -9521.025,E2 -9521.025} C_VEL
LIN {X 0,Y 432.387,Z 252.126,A -85,B 0,C 180,E1 -9523.955,E2 -9523.955} C_VEL
LIN {X 0,Y 432.458,Z 252.116,A -85,B 0,C 180,E1 -9527.799,E2 -9527.799} C_VEL
LIN {X 0,Y 432.459,Z 252.115,A -85,B 0,C 180,E1 -9531.585,E2 -9531.585} C_VEL
LIN {X 0,Y 432.547,Z 252.103,A -85,B 0,C 180,E1 -9534.4,E2 -9534.4} C_VEL
LIN {X 0,Y 432.587,Z 252.099,A -85,B 0,C 180,E1 -9538.133,E2 -9538.133} C_VEL
LIN {X 0,Y 432.611,Z 252.097,A -85,B 0,C 180,E1 -9539.995,E2 -9539.995} C_VEL
LIN {X 0,Y 432.571,Z 252.098,A -85,B 0,C 180,E1 -9542.788,E2 -9542.788} C_VEL
LIN {X 0,Y 432.572,Z 252.104,A -85,B 0,C 180,E1 -9545.588,E2 -9545.588} C_VEL
LIN {X 0,Y 432.449,Z 252.113,A -85,B 0,C 180,E1 -9548.405,E2 -9548.405} C_VEL
LIN {X 0,Y 432.441,Z 252.114,A -85,B 0,C 180,E1 -9552.191,E2 -9552.191} C_VEL
LIN {X 0,Y 432.408,Z 252.118,A -85,B 0,C 180,E1 -9556.033,E2 -9556.033} C_VEL
LIN {X 0,Y 432.363,Z 252.127,A -85,B 0,C 180,E1 -9559.479,E2 -9559.479} C_VEL
LIN {X 0,Y 432.291,Z 252.14,A -85,B 0,C 180,E1 -9562.958,E2 -9562.958} C_VEL
LIN {X 0,Y 432.332,Z 252.128,A -85,B 0,C 180,E1 -9566.027,E2 -9566.027} C_VEL
LIN {X 0,Y 432.31,Z 252.134,A -85,B 0,C 180,E1 -9569.182,E2 -9569.182} C_VEL
LIN {X 0,Y 432.287,Z 252.137,A -85,B 0,C 180,E1 -9572.437,E2 -9572.437} C_VEL
LIN {X 0,Y 432.307,Z 252.131,A -85,B 0,C 180,E1 -9575.626,E2 -9575.626} C_VEL
LIN {X 0,Y 432.292,Z 252.138,A -85,B 0,C 180,E1 -9578.708,E2 -9578.708} C_VEL
LIN {X 0,Y 432.327,Z 252.129,A -85,B 0,C 180,E1 -9581.787,E2 -9581.787} C_VEL
LIN {X 0,Y 432.333,Z 252.135,A -85,B 0,C 180,E1 -9584.336,E2 -9584.336} C_VEL
LIN {X 0,Y 432.318,Z 252.13,A -85,B 0,C 180,E1 -9587.004,E2 -9587.004} C_VEL
LIN {X 0,Y 432.308,Z 252.134,A -85,B 0,C 180,E1 -9589.812,E2 -9589.812} C_VEL
LIN {X 0,Y 432.264,Z 252.136,A -85,B 0,C 180,E1 -9593.019,E2 -9593.019} C_VEL
LIN {X 0,Y 432.305,Z 252.139,A -85,B 0,C 180,E1 -9595.992,E2 -9595.992} C_VEL
LIN {X 0,Y 432.338,Z 252.132,A -85,B 0,C 180,E1 -9599.74,E2 -9599.74} C_VEL
LIN {X 0,Y 432.341,Z 252.129,A -85,B 0,C 180,E1 -9603.369,E2 -9603.369} C_VEL
LIN {X 0,Y 432.32,Z 252.133,A -85,B 0,C 180,E1 -9606.021,E2 -9606.021} C_VEL
LIN {X 0,Y 432.315,Z 252.131,A -85,B 0,C 180,E1 -9609.045,E2 -9609.045} C_VEL
LIN {X 0,Y 432.321,Z 252.135,A -85,B 0,C 180,E1 -9612.009,E2 -9612.009} C_VEL
LIN {X 0,Y 432.348,Z 252.131,A -85,B 0,C 180,E1 -9614.925,E2 -9614.925} C_VEL
LIN {X 0,Y 432.419,Z 252.121,A -85,B 0,C 180,E1 -9617.803,E2 -9617.803} C_VEL
LIN {X 0,Y 432.432,Z 252.12,A -85,B 0,C 180,E1 -9621.589,E2 -9621.589} C_VEL
LIN {X 0,Y 432.542,Z 252.105,A -85,B 0,C 180,E1 -9624.406,E2 -9624.406} C_VEL
LIN {X 0,Y 432.541,Z 252.105,A -85,B 0,C 180,E1 -9628.138,E2 -9628.138} C_VEL
LIN {X 0,Y 432.668,Z 252.091,A -85,B 0,C 180,E1 -9630,E2 -9630} C_VEL
LIN {X 0,Y 432.548,Z 252.107,A -85,B 0,C 180,E1 -9632.794,E2 -9632.794} C_VEL
LIN {X 0,Y 432.402,Z 252.122,A -85,B 0,C 180,E1 -9634.992,E2 -9634.992} C_VEL
LIN {X 0,Y 431.844,Z 252.193,A -85,B 0,C 180,E1 -9635.77,E2 -9635.77} C_VEL
LIN {X 0,Y 429.011,Z 252.547,A -85,B 0,C 180,E1 -9637.035,E2 -9637.035} C_VEL
LIN {X 0,Y 426.535,Z 252.855,A -85,B 0,C 180,E1 -9638.057,E2 -9638.057} C_VEL
LIN {X 0,Y 425.451,Z 252.991,A -85,B 0,C 180,E1 -9638.846,E2 -9638.846} C_VEL
LIN {X 0,Y 425.356,Z 253,A -85,B 0,C 180,E1 -9639.114,E2 -9639.114} C_VEL
LIN {X 0,Y 425.341,Z 253.005,A -85,B 0,C 180,E1 -9642.912,E2 -9642.912} C_VEL
LIN {X 0,Y 425.307,Z 253.01,A -85,B 0,C 180,E1 -9646.611,E2 -9646.611} C_VEL
LIN {X 0,Y 425.301,Z 253.004,A -85,B 0,C 180,E1 -9649.651,E2 -9649.651} C_VEL
LIN {X 0,Y 425.277,Z 253.014,A -85,B 0,C 180,E1 -9652.339,E2 -9652.339} C_VEL
LIN {X 0,Y 425.242,Z 253.011,A -85,B 0,C 180,E1 -9655.448,E2 -9655.448} C_VEL
LIN {X 0,Y 425.28,Z 253.008,A -85,B 0,C 180,E1 -9658.635,E2 -9658.635} C_VEL
LIN {X 0,Y 425.218,Z 253.02,A -85,B 0,C 180,E1 -9661.93,E2 -9661.93} C_VEL
LIN {X 0,Y 425.246,Z 253.012,A -85,B 0,C 180,E1 -9665.34,E2 -9665.34} C_VEL
LIN {X 0,Y 425.262,Z 253.009,A -85,B 0,C 180,E1 -9669.05,E2 -9669.05} C_VEL
LIN {X 0,Y 425.284,Z 253.006,A -85,B 0,C 180,E1 -9672.651,E2 -9672.651} C_VEL
LIN {X 0,Y 425.274,Z 253.009,A -85,B 0,C 180,E1 -9676.057,E2 -9676.057} C_VEL
LIN {X 0,Y 425.258,Z 253.009,A -85,B 0,C 180,E1 -9678.63,E2 -9678.63} C_VEL
LIN {X 0,Y 425.251,Z 253.013,A -85,B 0,C 180,E1 -9681.106,E2 -9681.106} C_VEL
LIN {X 0,Y 425.262,Z 253.009,A -85,B 0,C 180,E1 -9684.67,E2 -9684.67} C_VEL
LIN {X 0,Y 425.229,Z 253.013,A -85,B 0,C 180,E1 -9688.079,E2 -9688.079} C_VEL
LIN {X 0,Y 425.299,Z 253.009,A -85,B 0,C 180,E1 -9691.374,E2 -9691.374} C_VEL
LIN {X 0,Y 425.324,Z 253.003,A -85,B 0,C 180,E1 -9693.511,E2 -9693.511} C_VEL
LIN {X 0,Y 425.258,Z 253.012,A -85,B 0,C 180,E1 -9696.64,E2 -9696.64} C_VEL
LIN {X 0,Y 425.27,Z 253.008,A -85,B 0,C 180,E1 -9699.7,E2 -9699.7} C_VEL
LIN {X 0,Y 425.311,Z 253.008,A -85,B 0,C 180,E1 -9702.703,E2 -9702.703} C_VEL
LIN {X 0,Y 425.325,Z 253.001,A -85,B 0,C 180,E1 -9705.656,E2 -9705.656} C_VEL
LIN {X 0,Y 425.332,Z 253.006,A -85,B 0,C 180,E1 -9708.57,E2 -9708.57} C_VEL
LIN {X 0,Y 425.492,Z 252.984,A -85,B 0,C 180,E1 -9712.316,E2 -9712.316} C_VEL
LIN {X 0,Y 425.529,Z 252.981,A -85,B 0,C 180,E1 -9714.319,E2 -9714.319} C_VEL
LIN {X 0,Y 425.561,Z 252.975,A -85,B 0,C 180,E1 -9718.113,E2 -9718.113} C_VEL
LIN {X 0,Y 425.501,Z 252.98,A -85,B 0,C 180,E1 -9720.952,E2 -9720.952} C_VEL
LIN {X 0,Y 425.506,Z 252.979,A -85,B 0,C 180,E1 -9722.846,E2 -9722.846} C_VEL
LIN {X 0,Y 425.472,Z 252.984,A -85,B 0,C 180,E1 -9726.645,E2 -9726.645} C_VEL
LIN {X 0,Y 425.391,Z 252.994,A -85,B 0,C 180,E1 -9729.515,E2 -9729.515} C_VEL
LIN {X 0,Y 425.394,Z 252.992,A -85,B 0,C 180,E1 -9732.908,E2 -9732.908} C_VEL
LIN {X 0,Y 425.315,Z 253.002,A -85,B 0,C 180,E1 -9736.587,E2 -9736.587} C_VEL
LIN {X 0,Y 425.331,Z 253.006,A -85,B 0,C 180,E1 -9739.639,E2 -9739.639} C_VEL
LIN {X 0,Y 425.291,Z 253.006,A -85,B 0,C 180,E1 -9742.343,E2 -9742.343} C_VEL
LIN {X 0,Y 425.264,Z 253.014,A -85,B 0,C 180,E1 -9745.452,E2 -9745.452} C_VEL
LIN {X 0,Y 425.307,Z 253.004,A -85,B 0,C 180,E1 -9748.862,E2 -9748.862} C_VEL
LIN {X 0,Y 425.267,Z 253.009,A -85,B 0,C 180,E1 -9751.931,E2 -9751.931} C_VEL
LIN {X 0,Y 425.302,Z 253.01,A -85,B 0,C 180,E1 -9755.34,E2 -9755.34} C_VEL
LIN {X 0,Y 425.288,Z 253.012,A -85,B 0,C 180,E1 -9758.904,E2 -9758.904} C_VEL
LIN {X 0,Y 425.305,Z 253.231,A -85,B 0,C 180,E1 -9760.525,E2 -9760.525} C_VEL
LIN {X 0,Y 425.823,Z 256.669,A -85,B 0,C 180,E1 -9763.887,E2 -9763.887} C_VEL
LIN {X 0,Y 426.241,Z 259.576,A -85,B 0,C 180,E1 -9766.514,E2 -9766.514} C_VEL
LIN {X 0,Y 426.339,Z 262.986,A -85,B 0,C 180,E1 -9769.318,E2 -9769.318} C_VEL
LIN {X 0,Y 426.21,Z 265.451,A -85,B 0,C 180,E1 -9771.201,E2 -9771.201} C_VEL
LIN {X 0,Y 425.751,Z 270.296,A -85,B 0,C 180,E1 -9774.708,E2 -9774.708} C_VEL
LIN {X 0,Y 425.47,Z 274.237,A -85,B 0,C 180,E1 -9777.402,E2 -9777.402} C_VEL
LIN {X 0,Y 425.193,Z 278.633,A -85,B 0,C 180,E1 -9780.274,E2 -9780.274} C_VEL
LIN {X 0,Y 424.954,Z 283.751,A -85,B 0,C 180,E1 -9783.479,E2 -9783.479} C_VEL
LIN {X 0,Y 424.658,Z 288.944,A -85,B 0,C 180,E1 -9786.598,E2 -9786.598} C_VEL
LIN {X 0,Y 424.498,Z 294.191,A -85,B 0,C 180,E1 -9789.655,E2 -9789.655} C_VEL
LIN {X 0,Y 424.324,Z 300.163,A -85,B 0,C 180,E1 -9793.019,E2 -9793.019} C_VEL
LIN {X 0,Y 427.076,Z 314.921,A -85,B 0,C 180,E1 -9793.606,E2 -9793.606} C_VEL
LIN {X 0,Y 428.684,Z 325.898,A -85,B 0,C 180,E1 -9794.184,E2 -9794.184} C_VEL
LIN {X 0,Y 428.025,Z 337.451,A -85,B 0,C 180,E1 -9794.891,E2 -9794.891} C_VEL
LIN {X 0,Y 427.457,Z 346.731,A -85,B 0,C 180,E1 -9795.601,E2 -9795.601} C_VEL
LIN {X 0,Y 426.963,Z 355.439,A -85,B 0,C 180,E1 -9796.408,E2 -9796.408} C_VEL
LIN {X 0,Y 426.402,Z 364.218,A -85,B 0,C 180,E1 -9797.386,E2 -9797.386} C_VEL
LIN {X 0,Y 425.881,Z 371.44,A -85,B 0,C 180,E1 -9798.337,E2 -9798.337} C_VEL
LIN {X 0,Y 425.431,Z 377.644,A -85,B 0,C 180,E1 -9799.29,E2 -9799.29} C_VEL
LIN {X 0,Y 425.024,Z 384.185,A -85,B 0,C 180,E1 -9800.482,E2 -9800.482} C_VEL
LIN {X 0,Y 424.744,Z 388.688,A -85,B 0,C 180,E1 -9801.436,E2 -9801.436} C_VEL
LIN {X 0,Y 424.451,Z 394.181,A -85,B 0,C 180,E1 -9802.867,E2 -9802.867} C_VEL
LIN {X 0,Y 424.252,Z 398.506,A -85,B 0,C 180,E1 -9804.296,E2 -9804.296} C_VEL
LIN {X 0,Y 424.223,Z 400.874,A -85,B 0,C 180,E1 -9805.249,E2 -9805.249} C_VEL
LIN {X 0,Y 424.13,Z 404.057,A -85,B 0,C 180,E1 -9807.151,E2 -9807.151} C_VEL
LIN {X 0,Y 424.131,Z 405.115,A -85,B 0,C 180,E1 -9808.101,E2 -9808.101} C_VEL
LIN {X 0,Y 424.075,Z 405.702,A -85,B 0,C 180,E1 -9809.05,E2 -9809.05} C_VEL
LIN {X 0,Y 424.075,Z 405.702,A -85,B 0,C 180,E1 -9810.95,E2 -9810.95} C_VEL
LIN {X 0,Y 424.131,Z 405.115,A -85,B 0,C 180,E1 -9811.899,E2 -9811.899} C_VEL
LIN {X 0,Y 424.112,Z 402.67,A -85,B 0,C 180,E1 -9813.801,E2 -9813.801} C_VEL
LIN {X 0,Y 424.247,Z 399.724,A -85,B 0,C 180,E1 -9815.227,E2 -9815.227} C_VEL
LIN {X 0,Y 424.372,Z 395.735,A -85,B 0,C 180,E1 -9816.657,E2 -9816.657} C_VEL
LIN {X 0,Y 424.598,Z 390.604,A -85,B 0,C 180,E1 -9818.088,E2 -9818.088} C_VEL
LIN {X 0,Y 424.925,Z 385.34,A -85,B 0,C 180,E1 -9819.28,E2 -9819.28} C_VEL
LIN {X 0,Y 425.336,Z 379.021,A -85,B 0,C 180,E1 -9820.472,E2 -9820.472} C_VEL
LIN {X 0,Y 425.729,Z 373.066,A -85,B 0,C 180,E1 -9821.426,E2 -9821.426} C_VEL
LIN {X 0,Y 426.258,Z 366.137,A -85,B 0,C 180,E1 -9822.377,E2 -9822.377} C_VEL
LIN {X 0,Y 426.772,Z 357.952,A -85,B 0,C 180,E1 -9823.329,E2 -9823.329} C_VEL
LIN {X 0,Y 427.224,Z 350.022,A -85,B 0,C 180,E1 -9824.111,E2 -9824.111} C_VEL
LIN {X 0,Y 427.848,Z 340.717,A -85,B 0,C 180,E1 -9824.872,E2 -9824.872} C_VEL
LIN {X 0,Y 428.379,Z 331.963,A -85,B 0,C 180,E1 -9825.462,E2 -9825.462} C_VEL
LIN {X 0,Y 428.557,Z 324.728,A -85,B 0,C 180,E1 -9825.882,E2 -9825.882} C_VEL
LIN {X 0,Y 426.609,Z 312.511,A -85,B 0,C 180,E1 -9826.497,E2 -9826.497} C_VEL
LIN {X 0,Y 424.484,Z 301.452,A -85,B 0,C 180,E1 -9826.922,E2 -9826.922} C_VEL
LIN {X 0,Y 424.323,Z 300.162,A -85,B 0,C 180,E1 -9826.981,E2 -9826.981} C_VEL
LIN {X 0,Y 424.495,Z 294.189,A -85,B 0,C 180,E1 -9830.345,E2 -9830.345} C_VEL
LIN {X 0,Y 424.661,Z 288.939,A -85,B 0,C 180,E1 -9833.402,E2 -9833.402} C_VEL
LIN {X 0,Y 424.979,Z 283.382,A -85,B 0,C 180,E1 -9836.74,E2 -9836.74} C_VEL
LIN {X 0,Y 425.198,Z 278.627,A -85,B 0,C 180,E1 -9839.726,E2 -9839.726} C_VEL
LIN {X 0,Y 425.519,Z 273.589,A -85,B 0,C 180,E1 -9843.027,E2 -9843.027} C_VEL
LIN {X 0,Y 425.856,Z 269.238,A -85,B 0,C 180,E1 -9846.03,E2 -9846.03} C_VEL
LIN {X 0,Y 426.257,Z 264.917,A -85,B 0,C 180,E1 -9849.198,E2 -9849.198} C_VEL
LIN {X 0,Y 426.341,Z 261.208,A -85,B 0,C 180,E1 -9852.111,E2 -9852.111} C_VEL
LIN {X 0,Y 426.067,Z 258.071,A -85,B 0,C 180,E1 -9854.819,E2 -9854.819} C_VEL
LIN {X 0,Y 425.502,Z 254.684,A -85,B 0,C 180,E1 -9858.009,E2 -9858.009} C_VEL
LIN {X 0,Y 425.252,Z 253.016,A -85,B 0,C 180,E1 -9859.865,E2 -9859.865} C_VEL
LIN {X 0,Y 425.282,Z 253.012,A -85,B 0,C 180,E1 -9862.486,E2 -9862.486} C_VEL
LIN {X 0,Y 425.293,Z 253.006,A -85,B 0,C 180,E1 -9865.812,E2 -9865.812} C_VEL
LIN {X 0,Y 425.296,Z 253.005,A -85,B 0,C 180,E1 -9869.236,E2 -9869.236} C_VEL
LIN {X 0,Y 425.253,Z 253.016,A -85,B 0,C 180,E1 -9872.431,E2 -9872.431} C_VEL
LIN {X 0,Y 425.325,Z 253.001,A -85,B 0,C 180,E1 -9875.596,E2 -9875.596} C_VEL
LIN {X 0,Y 425.293,Z 253.008,A -85,B 0,C 180,E1 -9878.677,E2 -9878.677} C_VEL
LIN {X 0,Y 425.307,Z 253.005,A -85,B 0,C 180,E1 -9881.697,E2 -9881.697} C_VEL
LIN {X 0,Y 425.303,Z 253.005,A -85,B 0,C 180,E1 -9884.664,E2 -9884.664} C_VEL
LIN {X 0,Y 425.412,Z 252.992,A -85,B 0,C 180,E1 -9887.593,E2 -9887.593} C_VEL
LIN {X 0,Y 425.404,Z 252.993,A -85,B 0,C 180,E1 -9891.444,E2 -9891.444} C_VEL
LIN {X 0,Y 425.505,Z 252.981,A -85,B 0,C 180,E1 -9894.307,E2 -9894.307} C_VEL
LIN {X 0,Y 425.556,Z 252.975,A -85,B 0,C 180,E1 -9898.102,E2 -9898.102} C_VEL
LIN {X 0,Y 425.563,Z 252.975,A -85,B 0,C 180,E1 -9899.994,E2 -9899.994} C_VEL
LIN {X 0,Y 425.524,Z 252.976,A -85,B 0,C 180,E1 -9902.834,E2 -9902.834} C_VEL
LIN {X 0,Y 425.491,Z 252.98,A -85,B 0,C 180,E1 -9906.583,E2 -9906.583} C_VEL
LIN {X 0,Y 425.382,Z 253,A -85,B 0,C 180,E1 -9909.504,E2 -9909.504} C_VEL
LIN {X 0,Y 425.376,Z 252.997,A -85,B 0,C 180,E1 -9912.897,E2 -9912.897} C_VEL
LIN {X 0,Y 425.34,Z 253,A -85,B 0,C 180,E1 -9916.598,E2 -9916.598} C_VEL
LIN {X 0,Y 425.304,Z 253.005,A -85,B 0,C 180,E1 -9919.629,E2 -9919.629} C_VEL
LIN {X 0,Y 425.262,Z 253.009,A -85,B 0,C 180,E1 -9922.333,E2 -9922.333} C_VEL
LIN {X 0,Y 425.262,Z 253.01,A -85,B 0,C 180,E1 -9925.44,E2 -9925.44} C_VEL
LIN {X 0,Y 425.318,Z 253.002,A -85,B 0,C 180,E1 -9927.552,E2 -9927.552} C_VEL
LIN {X 0,Y 425.254,Z 253.016,A -85,B 0,C 180,E1 -9930.81,E2 -9930.81} C_VEL
LIN {X 0,Y 425.275,Z 253.01,A -85,B 0,C 180,E1 -9934.282,E2 -9934.282} C_VEL
LIN {X 0,Y 425.237,Z 253.012,A -85,B 0,C 180,E1 -9937.689,E2 -9937.689} C_VEL
LIN {X 0,Y 425.24,Z 253.018,A -85,B 0,C 180,E1 -9940.515,E2 -9940.515} C_VEL
LIN {X 0,Y 425.272,Z 253.007,A -85,B 0,C 180,E1 -9943.354,E2 -9943.354} C_VEL
LIN {X 0,Y 425.285,Z 253.009,A -85,B 0,C 180,E1 -9946.634,E2 -9946.634} C_VEL
LIN {X 0,Y 425.261,Z 253.012,A -85,B 0,C 180,E1 -9949.871,E2 -9949.871} C_VEL
LIN {X 0,Y 425.234,Z 253.015,A -85,B 0,C 180,E1 -9952.483,E2 -9952.483} C_VEL
LIN {X 0,Y 425.253,Z 253.014,A -85,B 0,C 180,E1 -9955.813,E2 -9955.813} C_VEL
LIN {X 0,Y 425.248,Z 253.011,A -85,B 0,C 180,E1 -9959.232,E2 -9959.232} C_VEL
LIN {X 0,Y 425.292,Z 253.006,A -85,B 0,C 180,E1 -9962.439,E2 -9962.439} C_VEL
LIN {X 0,Y 425.298,Z 253.01,A -85,B 0,C 180,E1 -9965.599,E2 -9965.599} C_VEL
LIN {X 0,Y 425.268,Z 253.008,A -85,B 0,C 180,E1 -9968.681,E2 -9968.681} C_VEL
LIN {X 0,Y 425.275,Z 253.013,A -85,B 0,C 180,E1 -9971.701,E2 -9971.701} C_VEL
LIN {X 0,Y 425.301,Z 253.008,A -85,B 0,C 180,E1 -9974.669,E2 -9974.669} C_VEL
LIN {X 0,Y 425.368,Z 253.001,A -85,B 0,C 180,E1 -9977.597,E2 -9977.597} C_VEL
LIN {X 0,Y 425.402,Z 252.997,A -85,B 0,C 180,E1 -9981.449,E2 -9981.449} C_VEL
LIN {X 0,Y 425.52,Z 252.98,A -85,B 0,C 180,E1 -9984.313,E2 -9984.313} C_VEL
LIN {X 0,Y 425.511,Z 252.981,A -85,B 0,C 180,E1 -9988.107,E2 -9988.107} C_VEL
LIN {X 0,Y 425.638,Z 252.967,A -85,B 0,C 180,E1 -9990,E2 -9990} C_VEL
LIN {X 0,Y 425.5,Z 252.985,A -85,B 0,C 180,E1 -9992.84,E2 -9992.84} C_VEL
LIN {X 0,Y 425.52,Z 252.98,A -85,B 0,C 180,E1 -9995.687,E2 -9995.687} C_VEL
LIN {X 0,Y 425.402,Z 252.997,A -85,B 0,C 180,E1 -9998.551,E2 -9998.551} C_VEL
LIN {X 0,Y 425.356,Z 253,A -85,B 0,C 180,E1 -9999.114,E2 -9999.114} C_VEL
LIN {X 0,Y 424.674,Z 253.087,A -85,B 0,C 180,E1 -9999.904,E2 -9999.904} C_VEL
LIN {X 0,Y 421.823,Z 253.444,A -85,B 0,C 180,E1 -10001.188,E2 -10001.188} C_VEL
LIN {X 0,Y 419.412,Z 253.744,A -85,B 0,C 180,E1 -10002.224,E2 -10002.224} C_VEL
LIN {X 0,Y 418.365,Z 253.874,A -85,B 0,C 180,E1 -10003.025,E2 -10003.025} C_VEL
LIN {X 0,Y 418.273,Z 253.884,A -85,B 0,C 180,E1 -10003.297,E2 -10003.297} C_VEL
LIN {X 0,Y 418.258,Z 253.887,A -85,B 0,C 180,E1 -10006.741,E2 -10006.741} C_VEL
LIN {X 0,Y 418.242,Z 253.884,A -85,B 0,C 180,E1 -10009.805,E2 -10009.805} C_VEL
LIN {X 0,Y 418.23,Z 253.887,A -85,B 0,C 180,E1 -10012.736,E2 -10012.736} C_VEL
LIN {X 0,Y 418.215,Z 253.89,A -85,B 0,C 180,E1 -10015.907,E2 -10015.907} C_VEL
LIN {X 0,Y 418.217,Z 253.886,A -85,B 0,C 180,E1 -10019.165,E2 -10019.165} C_VEL
LIN {X 0,Y 418.205,Z 253.888,A -85,B 0,C 180,E1 -10022.849,E2 -10022.849} C_VEL
LIN {X 0,Y 418.196,Z 253.892,A -85,B 0,C 180,E1 -10026.243,E2 -10026.243} C_VEL
LIN {X 0,Y 418.216,Z 253.892,A -85,B 0,C 180,E1 -10029.685,E2 -10029.685} C_VEL
LIN {X 0,Y 418.237,Z 253.885,A -85,B 0,C 180,E1 -10032.334,E2 -10032.334} C_VEL
LIN {X 0,Y 418.229,Z 253.886,A -85,B 0,C 180,E1 -10035.119,E2 -10035.119} C_VEL
LIN {X 0,Y 418.247,Z 253.887,A -85,B 0,C 180,E1 -10037.778,E2 -10037.778} C_VEL
LIN {X 0,Y 418.204,Z 253.894,A -85,B 0,C 180,E1 -10041.563,E2 -10041.563} C_VEL
LIN {X 0,Y 418.222,Z 253.89,A -85,B 0,C 180,E1 -10045.165,E2 -10045.165} C_VEL
LIN {X 0,Y 418.21,Z 253.892,A -85,B 0,C 180,E1 -10047.478,E2 -10047.478} C_VEL
LIN {X 0,Y 418.237,Z 253.887,A -85,B 0,C 180,E1 -10050.902,E2 -10050.902} C_VEL
LIN {X 0,Y 418.239,Z 253.883,A -85,B 0,C 180,E1 -10054.102,E2 -10054.102} C_VEL
LIN {X 0,Y 418.206,Z 253.891,A -85,B 0,C 180,E1 -10057.27,E2 -10057.27} C_VEL
LIN {X 0,Y 418.259,Z 253.882,A -85,B 0,C 180,E1 -10060.37,E2 -10060.37} C_VEL
LIN {X 0,Y 418.295,Z 253.878,A -85,B 0,C 180,E1 -10063.411,E2 -10063.411} C_VEL
LIN {X 0,Y 418.329,Z 253.876,A -85,B 0,C 180,E1 -10067.006,E2 -10067.006} C_VEL
LIN {X 0,Y 418.322,Z 253.877,A -85,B 0,C 180,E1 -10070.334,E2 -10070.334} C_VEL
LIN {X 0,Y 418.455,Z 253.857,A -85,B 0,C 180,E1 -10073.254,E2 -10073.254} C_VEL
LIN {X 0,Y 418.317,Z 253.874,A -85,B 0,C 180,E1 -10075.187,E2 -10075.187} C_VEL
LIN {X 0,Y 418.53,Z 253.851,A -85,B 0,C 180,E1 -10078.081,E2 -10078.081} C_VEL
LIN {X 0,Y 418.464,Z 253.856,A -85,B 0,C 180,E1 -10080.968,E2 -10080.968} C_VEL
LIN {X 0,Y 418.463,Z 253.856,A -85,B 0,C 180,E1 -10082.893,E2 -10082.893} C_VEL
LIN {X 0,Y 418.465,Z 253.858,A -85,B 0,C 180,E1 -10085.789,E2 -10085.789} C_VEL
LIN {X 0,Y 418.374,Z 253.868,A -85,B 0,C 180,E1 -10088.701,E2 -10088.701} C_VEL
LIN {X 0,Y 418.312,Z 253.878,A -85,B 0,C 180,E1 -10091.636,E2 -10091.636} C_VEL
LIN {X 0,Y 418.279,Z 253.879,A -85,B 0,C 180,E1 -10094.603,E2 -10094.603} C_VEL
LIN {X 0,Y 418.249,Z 253.887,A -85,B 0,C 180,E1 -10097.61,E2 -10097.61} C_VEL
LIN {X 0,Y 418.25,Z 253.882,A -85,B 0,C 180,E1 -10100.668,E2 -10100.668} C_VEL
LIN {X 0,Y 418.261,Z 253.886,A -85,B 0,C 180,E1 -10103.787,E2 -10103.787} C_VEL
LIN {X 0,Y 418.213,Z 253.889,A -85,B 0,C 180,E1 -10107.046,E2 -10107.046} C_VEL
LIN {X 0,Y 418.246,Z 253.883,A -85,B 0,C 180,E1 -10110.276,E2 -10110.276} C_VEL
LIN {X 0,Y 418.24,Z 253.888,A -85,B 0,C 180,E1 -10113.682,E2 -10113.682} C_VEL
LIN {X 0,Y 418.245,Z 253.889,A -85,B 0,C 180,E1 -10117.228,E2 -10117.228} C_VEL
LIN {X 0,Y 418.209,Z 253.893,A -85,B 0,C 180,E1 -10119.691,E2 -10119.691} C_VEL
LIN {X 0,Y 418.583,Z 256.264,A -85,B 0,C 180,E1 -10122.375,E2 -10122.375} C_VEL
LIN {X 0,Y 419.062,Z 259.243,A -85,B 0,C 180,E1 -10125.222,E2 -10125.222} C_VEL
LIN {X 0,Y 419.337,Z 262.323,A -85,B 0,C 180,E1 -10127.904,E2 -10127.904} C_VEL
LIN {X 0,Y 419.267,Z 265.495,A -85,B 0,C 180,E1 -10130.455,E2 -10130.455} C_VEL
LIN {X 0,Y 418.848,Z 269.759,A -85,B 0,C 180,E1 -10133.654,E2 -10133.654} C_VEL
LIN {X 0,Y 418.45,Z 274.683,A -85,B 0,C 180,E1 -10137.12,E2 -10137.12} C_VEL
LIN {X 0,Y 418.172,Z 278.563,A -85,B 0,C 180,E1 -10139.723,E2 -10139.723} C_VEL
LIN {X 0,Y 417.939,Z 283.712,A -85,B 0,C 180,E1 -10143.035,E2 -10143.035} C_VEL
LIN {X 0,Y 417.603,Z 288.814,A -85,B 0,C 180,E1 -10146.178,E2 -10146.178} C_VEL
LIN {X 0,Y 417.441,Z 294.033,A -85,B 0,C 180,E1 -10149.296,E2 -10149.296} C_VEL
LIN {X 0,Y 417.259,Z 299.992,A -85,B 0,C 180,E1 -10152.731,E2 -10152.731} C_VEL
LIN {X 0,Y 419.887,Z 314.105,A -85,B 0,C 180,E1 -10153.296,E2 -10153.296} C_VEL
LIN {X 0,Y 421.753,Z 326.262,A -85,B 0,C 180,E1 -10153.951,E2 -10153.951} C_VEL
LIN {X 0,Y 421.147,Z 337.239,A -85,B 0,C 180,E1 -10154.638,E2 -10154.638} C_VEL
LIN {X 0,Y 420.558,Z 346.519,A -85,B 0,C 180,E1 -10155.36,E2 -10155.36} C_VEL
LIN {X 0,Y 419.997,Z 355.226,A -85,B 0,C 180,E1 -10156.179,E2 -10156.179} C_VEL
LIN {X 0,Y 419.45,Z 364.005,A -85,B 0,C 180,E1 -10157.173,E2 -10157.173} C_VEL
LIN {X 0,Y 418.916,Z 371.228,A -85,B 0,C 180,E1 -10158.141,E2 -10158.141} C_VEL
LIN {X 0,Y 418.42,Z 377.431,A -85,B 0,C 180,E1 -10159.108,E2 -10159.108} C_VEL
LIN {X 0,Y 417.97,Z 383.972,A -85,B 0,C 180,E1 -10160.32,E2 -10160.32} C_VEL
LIN {X 0,Y 417.702,Z 388.476,A -85,B 0,C 180,E1 -10161.29,E2 -10161.29} C_VEL
LIN {X 0,Y 417.377,Z 393.969,A -85,B 0,C 180,E1 -10162.745,E2 -10162.745} C_VEL
LIN {X 0,Y 417.164,Z 398.294,A -85,B 0,C 180,E1 -10164.199,E2 -10164.199} C_VEL
LIN {X 0,Y 417.133,Z 400.662,A -85,B 0,C 180,E1 -10165.168,E2 -10165.168} C_VEL
LIN {X 0,Y 417.028,Z 403.846,A -85,B 0,C 180,E1 -10167.102,E2 -10167.102} C_VEL
LIN {X 0,Y 417.059,Z 404.905,A -85,B 0,C 180,E1 -10168.069,E2 -10168.069} C_VEL
LIN {X 0,Y 416.999,Z 405.491,A -85,B 0,C 180,E1 -10169.034,E2 -10169.034} C_VEL
LIN {X 0,Y 416.999,Z 405.491,A -85,B 0,C 180,E1 -10170.966,E2 -10170.966} C_VEL
LIN {X 0,Y 417.059,Z 404.905,A -85,B 0,C 180,E1 -10171.931,E2 -10171.931} C_VEL
LIN {X 0,Y 417.028,Z 402.458,A -85,B 0,C 180,E1 -10173.865,E2 -10173.865} C_VEL
LIN {X 0,Y 417.165,Z 399.512,A -85,B 0,C 180,E1 -10175.316,E2 -10175.316} C_VEL
LIN {X 0,Y 417.288,Z 395.523,A -85,B 0,C 180,E1 -10176.77,E2 -10176.77} C_VEL
LIN {X 0,Y 417.558,Z 390.392,A -85,B 0,C 180,E1 -10178.225,E2 -10178.225} C_VEL
LIN {X 0,Y 417.893,Z 385.128,A -85,B 0,C 180,E1 -10179.437,E2 -10179.437} C_VEL
LIN {X 0,Y 418.307,Z 378.808,A -85,B 0,C 180,E1 -10180.65,E2 -10180.65} C_VEL
LIN {X 0,Y 418.76,Z 372.855,A -85,B 0,C 180,E1 -10181.618,E2 -10181.618} C_VEL
LIN {X 0,Y 419.29,Z 365.925,A -85,B 0,C 180,E1 -10182.586,E2 -10182.586} C_VEL
LIN {X 0,Y 419.842,Z 357.74,A -85,B 0,C 180,E1 -10183.553,E2 -10183.553} C_VEL
LIN {X 0,Y 420.378,Z 348.947,A -85,B 0,C 180,E1 -10184.425,E2 -10184.425} C_VEL
LIN {X 0,Y 420.961,Z 340.505,A -85,B 0,C 180,E1 -10185.121,E2 -10185.121} C_VEL
LIN {X 0,Y 421.532,Z 331.977,A -85,B 0,C 180,E1 -10185.705,E2 -10185.705} C_VEL
LIN {X 0,Y 421.625,Z 325.25,A -85,B 0,C 180,E1 -10186.112,E2 -10186.112} C_VEL
LIN {X 0,Y 419.578,Z 312.277,A -85,B 0,C 180,E1 -10186.782,E2 -10186.782} C_VEL
LIN {X 0,Y 417.471,Z 301.574,A -85,B 0,C 180,E1 -10187.207,E2 -10187.207} C_VEL
LIN {X 0,Y 417.259,Z 299.992,A -85,B 0,C 180,E1 -10187.269,E2 -10187.269} C_VEL
LIN {X 0,Y 417.38,Z 295.756,A -85,B 0,C 180,E1 -10189.68,E2 -10189.68} C_VEL
LIN {X 0,Y 417.549,Z 290.532,A -85,B 0,C 180,E1 -10192.775,E2 -10192.775} C_VEL
LIN {X 0,Y 417.789,Z 285.362,A -85,B 0,C 180,E1 -10195.936,E2 -10195.936} C_VEL
LIN {X 0,Y 418.102,Z 280.242,A -85,B 0,C 180,E1 -10199.174,E2 -10199.174} C_VEL
LIN {X 0,Y 418.425,Z 275.203,A -85,B 0,C 180,E1 -10202.512,E2 -10202.512} C_VEL
LIN {X 0,Y 418.803,Z 270.283,A -85,B 0,C 180,E1 -10205.968,E2 -10205.968} C_VEL
LIN {X 0,Y 419.114,Z 267.059,A -85,B 0,C 180,E1 -10208.348,E2 -10208.348} C_VEL
LIN {X 0,Y 419.331,Z 263.594,A -85,B 0,C 180,E1 -10211.04,E2 -10211.04} C_VEL
LIN {X 0,Y 419.278,Z 260.781,A -85,B 0,C 180,E1 -10213.412,E2 -10213.412} C_VEL
LIN {X 0,Y 418.756,Z 257.389,A -85,B 0,C 180,E1 -10216.515,E2 -10216.515} C_VEL
LIN {X 0,Y 418.36,Z 254.784,A -85,B 0,C 180,E1 -10219.107,E2 -10219.107} C_VEL
LIN {X 0,Y 418.215,Z 253.892,A -85,B 0,C 180,E1 -10220.624,E2 -10220.624} C_VEL
LIN {X 0,Y 418.248,Z 253.883,A -85,B 0,C 180,E1 -10223.972,E2 -10223.972} C_VEL
LIN {X 0,Y 418.258,Z 253.883,A -85,B 0,C 180,E1 -10227.154,E2 -10227.154} C_VEL
LIN {X 0,Y 418.264,Z 253.884,A -85,B 0,C 180,E1 -10230.834,E2 -10230.834} C_VEL
LIN {X 0,Y 418.224,Z 253.888,A -85,B 0,C 180,E1 -10234.088,E2 -10234.088} C_VEL
LIN {X 0,Y 418.232,Z 253.884,A -85,B 0,C 180,E1 -10237.259,E2 -10237.259} C_VEL
LIN {X 0,Y 418.286,Z 253.884,A -85,B 0,C 180,E1 -10240.36,E2 -10240.36} C_VEL
LIN {X 0,Y 418.281,Z 253.878,A -85,B 0,C 180,E1 -10243.398,E2 -10243.398} C_VEL
LIN {X 0,Y 418.347,Z 253.87,A -85,B 0,C 180,E1 -10246.995,E2 -10246.995} C_VEL
LIN {X 0,Y 418.333,Z 253.875,A -85,B 0,C 180,E1 -10250.323,E2 -10250.323} C_VEL
LIN {X 0,Y 418.437,Z 253.86,A -85,B 0,C 180,E1 -10253.243,E2 -10253.243} C_VEL
LIN {X 0,Y 418.309,Z 253.875,A -85,B 0,C 180,E1 -10255.176,E2 -10255.176} C_VEL
LIN {X 0,Y 418.525,Z 253.851,A -85,B 0,C 180,E1 -10258.07,E2 -10258.07} C_VEL
LIN {X 0,Y 418.398,Z 253.864,A -85,B 0,C 180,E1 -10260.957,E2 -10260.957} C_VEL
LIN {X 0,Y 418.48,Z 253.854,A -85,B 0,C 180,E1 -10262.882,E2 -10262.882} C_VEL
LIN {X 0,Y 418.452,Z 253.857,A -85,B 0,C 180,E1 -10266.584,E2 -10266.584} C_VEL
LIN {X 0,Y 418.322,Z 253.877,A -85,B 0,C 180,E1 -10269.666,E2 -10269.666} C_VEL
LIN {X 0,Y 418.329,Z 253.876,A -85,B 0,C 180,E1 -10272.994,E2 -10272.994} C_VEL
LIN {X 0,Y 418.291,Z 253.879,A -85,B 0,C 180,E1 -10276.729,E2 -10276.729} C_VEL
LIN {X 0,Y 418.246,Z 253.883,A -85,B 0,C 180,E1 -10279.784,E2 -10279.784} C_VEL
LIN {X 0,Y 418.206,Z 253.891,A -85,B 0,C 180,E1 -10282.73,E2 -10282.73} C_VEL
LIN {X 0,Y 418.239,Z 253.883,A -85,B 0,C 180,E1 -10285.898,E2 -10285.898} C_VEL
LIN {X 0,Y 418.233,Z 253.887,A -85,B 0,C 180,E1 -10289.156,E2 -10289.156} C_VEL
LIN {X 0,Y 418.222,Z 253.891,A -85,B 0,C 180,E1 -10292.838,E2 -10292.838} C_VEL
LIN {X 0,Y 418.207,Z 253.89,A -85,B 0,C 180,E1 -10296.232,E2 -10296.232} C_VEL
LIN {X 0,Y 418.202,Z 253.888,A -85,B 0,C 180,E1 -10299.677,E2 -10299.677} C_VEL
LIN {X 0,Y 418.24,Z 253.889,A -85,B 0,C 180,E1 -10302.324,E2 -10302.324} C_VEL
LIN {X 0,Y 418.229,Z 253.885,A -85,B 0,C 180,E1 -10305.109,E2 -10305.109} C_VEL
LIN {X 0,Y 418.244,Z 253.885,A -85,B 0,C 180,E1 -10307.768,E2 -10307.768} C_VEL
LIN {X 0,Y 418.215,Z 253.888,A -85,B 0,C 180,E1 -10311.555,E2 -10311.555} C_VEL
LIN {X 0,Y 418.206,Z 253.888,A -85,B 0,C 180,E1 -10315.155,E2 -10315.155} C_VEL
LIN {X 0,Y 418.194,Z 253.891,A -85,B 0,C 180,E1 -10317.468,E2 -10317.468} C_VEL
LIN {X 0,Y 418.219,Z 253.886,A -85,B 0,C 180,E1 -10320.89,E2 -10320.89} C_VEL
LIN {X 0,Y 418.215,Z 253.89,A -85,B 0,C 180,E1 -10324.093,E2 -10324.093} C_VEL
LIN {X 0,Y 418.237,Z 253.889,A -85,B 0,C 180,E1 -10327.527,E2 -10327.527} C_VEL
LIN {X 0,Y 418.256,Z 253.884,A -85,B 0,C 180,E1 -10330.363,E2 -10330.363} C_VEL
LIN {X 0,Y 418.263,Z 253.887,A -85,B 0,C 180,E1 -10333.403,E2 -10333.403} C_VEL
LIN {X 0,Y 418.292,Z 253.883,A -85,B 0,C 180,E1 -10336.992,E2 -10336.992} C_VEL
LIN {X 0,Y 418.303,Z 253.88,A -85,B 0,C 180,E1 -10340.328,E2 -10340.328} C_VEL
LIN {X 0,Y 418.451,Z 253.862,A -85,B 0,C 180,E1 -10343.248,E2 -10343.248} C_VEL
LIN {X 0,Y 418.285,Z 253.884,A -85,B 0,C 180,E1 -10345.181,E2 -10345.181} C_VEL
LIN {X 0,Y 418.48,Z 253.857,A -85,B 0,C 180,E1 -10348.075,E2 -10348.075} C_VEL
LIN {X 0,Y 418.608,Z 253.843,A -85,B 0,C 180,E1 -10350,E2 -10350} C_VEL
LIN {X 0,Y 418.454,Z 253.862,A -85,B 0,C 180,E1 -10352.888,E2 -10352.888} C_VEL
LIN {X 0,Y 418.477,Z 253.858,A -85,B 0,C 180,E1 -10355.783,E2 -10355.783} C_VEL
LIN {X 0,Y 418.353,Z 253.876,A -85,B 0,C 180,E1 -10358.696,E2 -10358.696} C_VEL
LIN {X 0,Y 418.308,Z 253.882,A -85,B 0,C 180,E1 -10362.616,E2 -10362.616} C_VEL
LIN {X 0,Y 418.273,Z 253.884,A -85,B 0,C 180,E1 -10363.297,E2 -10363.297} C_VEL
LIN {X 0,Y 417.582,Z 253.971,A -85,B 0,C 180,E1 -10364.1,E2 -10364.1} C_VEL
LIN {X 0,Y 414.704,Z 254.328,A -85,B 0,C 180,E1 -10365.406,E2 -10365.406} C_VEL
LIN {X 0,Y 412.286,Z 254.632,A -85,B 0,C 180,E1 -10366.46,E2 -10366.46} C_VEL
LIN {X 0,Y 411.259,Z 254.757,A -85,B 0,C 180,E1 -10367.275,E2 -10367.275} C_VEL
LIN {X 0,Y 411.181,Z 254.766,A -85,B 0,C 180,E1 -10367.551,E2 -10367.551} C_VEL
LIN {X 0,Y 411.181,Z 254.763,A -85,B 0,C 180,E1 -10371.034,E2 -10371.034} C_VEL
LIN {X 0,Y 411.173,Z 254.77,A -85,B 0,C 180,E1 -10374.218,E2 -10374.218} C_VEL
LIN {X 0,Y 411.202,Z 254.761,A -85,B 0,C 180,E1 -10377.481,E2 -10377.481} C_VEL
LIN {X 0,Y 411.145,Z 254.767,A -85,B 0,C 180,E1 -10380.851,E2 -10380.851} C_VEL
LIN {X 0,Y 411.152,Z 254.769,A -85,B 0,C 180,E1 -10384.338,E2 -10384.338} C_VEL
LIN {X 0,Y 411.153,Z 254.772,A -85,B 0,C 180,E1 -10387.977,E2 -10387.977} C_VEL
LIN {X 0,Y 411.161,Z 254.767,A -85,B 0,C 180,E1 -10391.241,E2 -10391.241} C_VEL
LIN {X 0,Y 411.191,Z 254.762,A -85,B 0,C 180,E1 -10394.487,E2 -10394.487} C_VEL
LIN {X 0,Y 411.184,Z 254.766,A -85,B 0,C 180,E1 -10397.303,E2 -10397.303} C_VEL
LIN {X 0,Y 411.167,Z 254.765,A -85,B 0,C 180,E1 -10400.78,E2 -10400.78} C_VEL
LIN {X 0,Y 411.16,Z 254.765,A -85,B 0,C 180,E1 -10404.477,E2 -10404.477} C_VEL
LIN {X 0,Y 411.172,Z 254.766,A -85,B 0,C 180,E1 -10406.879,E2 -10406.879} C_VEL
LIN {X 0,Y 411.201,Z 254.762,A -85,B 0,C 180,E1 -10410.65,E2 -10410.65} C_VEL
LIN {X 0,Y 411.208,Z 254.761,A -85,B 0,C 180,E1 -10413.625,E2 -10413.625} C_VEL
LIN {X 0,Y 411.169,Z 254.769,A -85,B 0,C 180,E1 -10416.858,E2 -10416.858} C_VEL
LIN {X 0,Y 411.19,Z 254.762,A -85,B 0,C 180,E1 -10420.057,E2 -10420.057} C_VEL
LIN {X 0,Y 411.243,Z 254.758,A -85,B 0,C 180,E1 -10423.137,E2 -10423.137} C_VEL
LIN {X 0,Y 411.288,Z 254.754,A -85,B 0,C 180,E1 -10426.902,E2 -10426.902} C_VEL
LIN {X 0,Y 411.274,Z 254.753,A -85,B 0,C 180,E1 -10430.167,E2 -10430.167} C_VEL
LIN {X 0,Y 411.42,Z 254.734,A -85,B 0,C 180,E1 -10433.139,E2 -10433.139} C_VEL
LIN {X 0,Y 411.289,Z 254.75,A -85,B 0,C 180,E1 -10435.105,E2 -10435.105} C_VEL
LIN {X 0,Y 411.499,Z 254.726,A -85,B 0,C 180,E1 -10438.048,E2 -10438.048} C_VEL
LIN {X 0,Y 411.428,Z 254.732,A -85,B 0,C 180,E1 -10440.984,E2 -10440.984} C_VEL
LIN {X 0,Y 411.422,Z 254.733,A -85,B 0,C 180,E1 -10442.943,E2 -10442.943} C_VEL
LIN {X 0,Y 411.386,Z 254.737,A -85,B 0,C 180,E1 -10446.874,E2 -10446.874} C_VEL
LIN {X 0,Y 411.286,Z 254.755,A -85,B 0,C 180,E1 -10449.844,E2 -10449.844} C_VEL
LIN {X 0,Y 411.306,Z 254.747,A -85,B 0,C 180,E1 -10453.109,E2 -10453.109} C_VEL
LIN {X 0,Y 411.21,Z 254.759,A -85,B 0,C 180,E1 -10456.896,E2 -10456.896} C_VEL
LIN {X 0,Y 411.214,Z 254.762,A -85,B 0,C 180,E1 -10459.992,E2 -10459.992} C_VEL
LIN {X 0,Y 411.192,Z 254.763,A -85,B 0,C 180,E1 -10463.153,E2 -10463.153} C_VEL
LIN {X 0,Y 411.177,Z 254.763,A -85,B 0,C 180,E1 -10466.39,E2 -10466.39} C_VEL
LIN {X 0,Y 411.202,Z 254.764,A -85,B 0,C 180,E1 -10469.717,E2 -10469.717} C_VEL
LIN {X 0,Y 411.213,Z 254.764,A -85,B 0,C 180,E1 -10473.16,E2 -10473.16} C_VEL
LIN {X 0,Y 411.2,Z 254.765,A -85,B 0,C 180,E1 -10476.555,E2 -10476.555} C_VEL
LIN {X 0,Y 411.178,Z 254.891,A -85,B 0,C 180,E1 -10479.723,E2 -10479.723} C_VEL
LIN {X 0,Y 411.684,Z 258.131,A -85,B 0,C 180,E1 -10483.071,E2 -10483.071} C_VEL
LIN {X 0,Y 412.114,Z 260.956,A -85,B 0,C 180,E1 -10485.75,E2 -10485.75} C_VEL
LIN {X 0,Y 412.317,Z 264.21,A -85,B 0,C 180,E1 -10488.594,E2 -10488.594} C_VEL
LIN {X 0,Y 412.077,Z 268.08,A -85,B 0,C 180,E1 -10491.682,E2 -10491.682} C_VEL
LIN {X 0,Y 411.65,Z 272.609,A -85,B 0,C 180,E1 -10495.039,E2 -10495.039} C_VEL
LIN {X 0,Y 411.275,Z 276.829,A -85,B 0,C 180,E1 -10498.013,E2 -10498.013} C_VEL
LIN {X 0,Y 410.965,Z 281.865,A -85,B 0,C 180,E1 -10501.391,E2 -10501.391} C_VEL
LIN {X 0,Y 410.661,Z 286.969,A -85,B 0,C 180,E1 -10504.669,E2 -10504.669} C_VEL
LIN {X 0,Y 410.453,Z 292.149,A -85,B 0,C 180,E1 -10507.871,E2 -10507.871} C_VEL
LIN {X 0,Y 410.254,Z 297.377,A -85,B 0,C 180,E1 -10511.005,E2 -10511.005} C_VEL
LIN {X 0,Y 410.181,Z 300.005,A -85,B 0,C 180,E1 -10512.445,E2 -10512.445} C_VEL
LIN {X 0,Y 412.237,Z 310.477,A -85,B 0,C 180,E1 -10512.853,E2 -10512.853} C_VEL
LIN {X 0,Y 413.835,Z 320.158,A -85,B 0,C 180,E1 -10513.335,E2 -10513.335} C_VEL
LIN {X 0,Y 414.808,Z 326.63,A -85,B 0,C 180,E1 -10513.712,E2 -10513.712} C_VEL
LIN {X 0,Y 414.295,Z 337.027,A -85,B 0,C 180,E1 -10514.378,E2 -10514.378} C_VEL
LIN {X 0,Y 413.663,Z 346.307,A -85,B 0,C 180,E1 -10515.11,E2 -10515.11} C_VEL
LIN {X 0,Y 413.041,Z 355.459,A -85,B 0,C 180,E1 -10515.99,E2 -10515.99} C_VEL
LIN {X 0,Y 412.488,Z 363.793,A -85,B 0,C 180,E1 -10516.953,E2 -10516.953} C_VEL
LIN {X 0,Y 411.945,Z 371.016,A -85,B 0,C 180,E1 -10517.937,E2 -10517.937} C_VEL
LIN {X 0,Y 411.426,Z 377.219,A -85,B 0,C 180,E1 -10518.921,E2 -10518.921} C_VEL
LIN {X 0,Y 410.93,Z 383.759,A -85,B 0,C 180,E1 -10520.153,E2 -10520.153} C_VEL
LIN {X 0,Y 410.642,Z 388.264,A -85,B 0,C 180,E1 -10521.14,E2 -10521.14} C_VEL
LIN {X 0,Y 410.304,Z 393.757,A -85,B 0,C 180,E1 -10522.619,E2 -10522.619} C_VEL
LIN {X 0,Y 410.089,Z 398.082,A -85,B 0,C 180,E1 -10524.098,E2 -10524.098} C_VEL
LIN {X 0,Y 410.047,Z 400.45,A -85,B 0,C 180,E1 -10525.084,E2 -10525.084} C_VEL
LIN {X 0,Y 409.947,Z 402.247,A -85,B 0,C 180,E1 -10526.068,E2 -10526.068} C_VEL
LIN {X 0,Y 409.97,Z 404.694,A -85,B 0,C 180,E1 -10528.035,E2 -10528.035} C_VEL
LIN {X 0,Y 409.925,Z 405.281,A -85,B 0,C 180,E1 -10529.018,E2 -10529.018} C_VEL
LIN {X 0,Y 409.925,Z 405.281,A -85,B 0,C 180,E1 -10530.982,E2 -10530.982} C_VEL
LIN {X 0,Y 409.97,Z 404.694,A -85,B 0,C 180,E1 -10531.965,E2 -10531.965} C_VEL
LIN {X 0,Y 409.947,Z 402.247,A -85,B 0,C 180,E1 -10533.932,E2 -10533.932} C_VEL
LIN {X 0,Y 410.064,Z 399.3,A -85,B 0,C 180,E1 -10535.409,E2 -10535.409} C_VEL
LIN {X 0,Y 410.212,Z 395.311,A -85,B 0,C 180,E1 -10536.888,E2 -10536.888} C_VEL
LIN {X 0,Y 410.508,Z 390.18,A -85,B 0,C 180,E1 -10538.367,E2 -10538.367} C_VEL
LIN {X 0,Y 410.861,Z 384.916,A -85,B 0,C 180,E1 -10539.6,E2 -10539.6} C_VEL
LIN {X 0,Y 411.286,Z 378.595,A -85,B 0,C 180,E1 -10540.834,E2 -10540.834} C_VEL
LIN {X 0,Y 411.793,Z 372.643,A -85,B 0,C 180,E1 -10541.818,E2 -10541.818} C_VEL
LIN {X 0,Y 412.33,Z 365.713,A -85,B 0,C 180,E1 -10542.802,E2 -10542.802} C_VEL
LIN {X 0,Y 412.911,Z 357.528,A -85,B 0,C 180,E1 -10543.785,E2 -10543.785} C_VEL
LIN {X 0,Y 413.475,Z 348.872,A -85,B 0,C 180,E1 -10544.658,E2 -10544.658} C_VEL
LIN {X 0,Y 414.102,Z 340.293,A -85,B 0,C 180,E1 -10545.377,E2 -10545.377} C_VEL
LIN {X 0,Y 414.67,Z 332.014,A -85,B 0,C 180,E1 -10545.957,E2 -10545.957} C_VEL
LIN {X 0,Y 414.792,Z 326.673,A -85,B 0,C 180,E1 -10546.286,E2 -10546.286} C_VEL
LIN {X 0,Y 412.7,Z 313.167,A -85,B 0,C 180,E1 -10547.03,E2 -10547.03} C_VEL
LIN {X 0,Y 410.465,Z 301.728,A -85,B 0,C 180,E1 -10547.501,E2 -10547.501} C_VEL
LIN {X 0,Y 410.165,Z 299.808,A -85,B 0,C 180,E1 -10547.577,E2 -10547.577} C_VEL
LIN {X 0,Y 410.298,Z 295.595,A -85,B 0,C 180,E1 -10550.034,E2 -10550.034} C_VEL
LIN {X 0,Y 410.482,Z 290.403,A -85,B 0,C 180,E1 -10553.19,E2 -10553.19} C_VEL
LIN {X 0,Y 410.768,Z 285.252,A -85,B 0,C 180,E1 -10556.413,E2 -10556.413} C_VEL
LIN {X 0,Y 411.074,Z 280.157,A -85,B 0,C 180,E1 -10559.722,E2 -10559.722} C_VEL
LIN {X 0,Y 411.433,Z 275.116,A -85,B 0,C 180,E1 -10563.17,E2 -10563.17} C_VEL
LIN {X 0,Y 411.857,Z 270.279,A -85,B 0,C 180,E1 -10566.672,E2 -10566.672} C_VEL
LIN {X 0,Y 412.148,Z 267.053,A -85,B 0,C 180,E1 -10569.118,E2 -10569.118} C_VEL
LIN {X 0,Y 412.308,Z 263.902,A -85,B 0,C 180,E1 -10571.664,E2 -10571.664} C_VEL
LIN {X 0,Y 412.13,Z 260.831,A -85,B 0,C 180,E1 -10574.359,E2 -10574.359} C_VEL
LIN {X 0,Y 411.636,Z 257.823,A -85,B 0,C 180,E1 -10577.235,E2 -10577.235} C_VEL
LIN {X 0,Y 411.178,Z 254.888,A -85,B 0,C 180,E1 -10580.277,E2 -10580.277} C_VEL
LIN {X 0,Y 411.199,Z 254.762,A -85,B 0,C 180,E1 -10583.445,E2 -10583.445} C_VEL
LIN {X 0,Y 411.214,Z 254.763,A -85,B 0,C 180,E1 -10586.87,E2 -10586.87} C_VEL
LIN {X 0,Y 411.216,Z 254.764,A -85,B 0,C 180,E1 -10590.646,E2 -10590.646} C_VEL
LIN {X 0,Y 411.177,Z 254.763,A -85,B 0,C 180,E1 -10593.61,E2 -10593.61} C_VEL
LIN {X 0,Y 411.192,Z 254.763,A -85,B 0,C 180,E1 -10596.847,E2 -10596.847} C_VEL
LIN {X 0,Y 411.216,Z 254.762,A -85,B 0,C 180,E1 -10600.047,E2 -10600.047} C_VEL
LIN {X 0,Y 411.222,Z 254.758,A -85,B 0,C 180,E1 -10603.147,E2 -10603.147} C_VEL
LIN {X 0,Y 411.306,Z 254.747,A -85,B 0,C 180,E1 -10606.891,E2 -10606.891} C_VEL
LIN {X 0,Y 411.286,Z 254.755,A -85,B 0,C 180,E1 -10610.156,E2 -10610.156} C_VEL
LIN {X 0,Y 411.386,Z 254.737,A -85,B 0,C 180,E1 -10613.126,E2 -10613.126} C_VEL
LIN {X 0,Y 411.281,Z 254.751,A -85,B 0,C 180,E1 -10615.093,E2 -10615.093} C_VEL
LIN {X 0,Y 411.494,Z 254.727,A -85,B 0,C 180,E1 -10618.037,E2 -10618.037} C_VEL
LIN {X 0,Y 411.368,Z 254.74,A -85,B 0,C 180,E1 -10620.973,E2 -10620.973} C_VEL
LIN {X 0,Y 411.437,Z 254.732,A -85,B 0,C 180,E1 -10622.932,E2 -10622.932} C_VEL
LIN {X 0,Y 411.42,Z 254.734,A -85,B 0,C 180,E1 -10626.861,E2 -10626.861} C_VEL
LIN {X 0,Y 411.274,Z 254.753,A -85,B 0,C 180,E1 -10629.833,E2 -10629.833} C_VEL
LIN {X 0,Y 411.288,Z 254.754,A -85,B 0,C 180,E1 -10633.098,E2 -10633.098} C_VEL
LIN {X 0,Y 411.237,Z 254.759,A -85,B 0,C 180,E1 -10636.883,E2 -10636.883} C_VEL
LIN {X 0,Y 411.207,Z 254.759,A -85,B 0,C 180,E1 -10639.981,E2 -10639.981} C_VEL
LIN {X 0,Y 411.169,Z 254.769,A -85,B 0,C 180,E1 -10643.142,E2 -10643.142} C_VEL
LIN {X 0,Y 411.208,Z 254.761,A -85,B 0,C 180,E1 -10646.375,E2 -10646.375} C_VEL
LIN {X 0,Y 411.168,Z 254.764,A -85,B 0,C 180,E1 -10649.707,E2 -10649.707} C_VEL
LIN {X 0,Y 411.171,Z 254.766,A -85,B 0,C 180,E1 -10653.15,E2 -10653.15} C_VEL
LIN {X 0,Y 411.154,Z 254.773,A -85,B 0,C 180,E1 -10656.547,E2 -10656.547} C_VEL
LIN {X 0,Y 411.166,Z 254.765,A -85,B 0,C 180,E1 -10659.721,E2 -10659.721} C_VEL
LIN {X 0,Y 411.177,Z 254.764,A -85,B 0,C 180,E1 -10663.122,E2 -10663.122} C_VEL
LIN {X 0,Y 411.194,Z 254.763,A -85,B 0,C 180,E1 -10665.866,E2 -10665.866} C_VEL
LIN {X 0,Y 411.164,Z 254.765,A -85,B 0,C 180,E1 -10669.495,E2 -10669.495} C_VEL
LIN {X 0,Y 411.153,Z 254.772,A -85,B 0,C 180,E1 -10672.023,E2 -10672.023} C_VEL
LIN {X 0,Y 411.152,Z 254.769,A -85,B 0,C 180,E1 -10675.662,E2 -10675.662} C_VEL
LIN {X 0,Y 411.145,Z 254.767,A -85,B 0,C 180,E1 -10679.149,E2 -10679.149} C_VEL
LIN {X 0,Y 411.202,Z 254.761,A -85,B 0,C 180,E1 -10682.519,E2 -10682.519} C_VEL
LIN {X 0,Y 411.173,Z 254.77,A -85,B 0,C 180,E1 -10685.782,E2 -10685.782} C_VEL
LIN {X 0,Y 411.181,Z 254.763,A -85,B 0,C 180,E1 -10688.966,E2 -10688.966} C_VEL
LIN {X 0,Y 411.193,Z 254.766,A -85,B 0,C 180,E1 -10692.083,E2 -10692.083} C_VEL
LIN {X 0,Y 411.21,Z 254.765,A -85,B 0,C 180,E1 -10695.146,E2 -10695.146} C_VEL
LIN {X 0,Y 411.238,Z 254.758,A -85,B 0,C 180,E1 -10698.166,E2 -10698.166} C_VEL
LIN {X 0,Y 411.418,Z 254.738,A -85,B 0,C 180,E1 -10702.146,E2 -10702.146} C_VEL
LIN {X 0,Y 411.437,Z 254.735,A -85,B 0,C 180,E1 -10704.118,E2 -10704.118} C_VEL
LIN {X 0,Y 411.45,Z 254.733,A -85,B 0,C 180,E1 -10708.042,E2 -10708.042} C_VEL
LIN {X 0,Y 411.578,Z 254.719,A -85,B 0,C 180,E1 -10710,E2 -10710} C_VEL
LIN {X 0,Y 411.41,Z 254.739,A -85,B 0,C 180,E1 -10712.938,E2 -10712.938} C_VEL
LIN {X 0,Y 411.437,Z 254.735,A -85,B 0,C 180,E1 -10715.882,E2 -10715.882} C_VEL
LIN {X 0,Y 411.305,Z 254.753,A -85,B 0,C 180,E1 -10718.846,E2 -10718.846} C_VEL
LIN {X 0,Y 411.238,Z 254.758,A -85,B 0,C 180,E1 -10721.834,E2 -10721.834} C_VEL
LIN {X 0,Y 411.21,Z 254.765,A -85,B 0,C 180,E1 -10724.854,E2 -10724.854} C_VEL
LIN {X 0,Y 411.181,Z 254.766,A -85,B 0,C 180,E1 -10727.551,E2 -10727.551} C_VEL
LIN {X 0,Y 410.523,Z 254.851,A -85,B 0,C 180,E1 -10728.37,E2 -10728.37} C_VEL
LIN {X 0,Y 407.662,Z 255.203,A -85,B 0,C 180,E1 -10729.699,E2 -10729.699} C_VEL
LIN {X 0,Y 405.241,Z 255.505,A -85,B 0,C 180,E1 -10730.773,E2 -10730.773} C_VEL
LIN {X 0,Y 404.212,Z 255.631,A -85,B 0,C 180,E1 -10731.603,E2 -10731.603} C_VEL
LIN {X 0,Y 404.135,Z 255.64,A -85,B 0,C 180,E1 -10731.884,E2 -10731.884} C_VEL
LIN {X 0,Y 404.158,Z 255.637,A -85,B 0,C 180,E1 -10735.3,E2 -10735.3} C_VEL
LIN {X 0,Y 404.141,Z 255.645,A -85,B 0,C 180,E1 -10738.003,E2 -10738.003} C_VEL
LIN {X 0,Y 404.091,Z 255.648,A -85,B 0,C 180,E1 -10741.564,E2 -10741.564} C_VEL
LIN {X 0,Y 404.132,Z 255.641,A -85,B 0,C 180,E1 -10745.021,E2 -10745.021} C_VEL
LIN {X 0,Y 404.113,Z 255.643,A -85,B 0,C 180,E1 -10748.761,E2 -10748.761} C_VEL
LIN {X 0,Y 404.143,Z 255.645,A -85,B 0,C 180,E1 -10751.616,E2 -10751.616} C_VEL
LIN {X 0,Y 404.155,Z 255.638,A -85,B 0,C 180,E1 -10754.535,E2 -10754.535} C_VEL
LIN {X 0,Y 404.162,Z 255.641,A -85,B 0,C 180,E1 -10757.31,E2 -10757.31} C_VEL
LIN {X 0,Y 404.128,Z 255.643,A -85,B 0,C 180,E1 -10759.961,E2 -10759.961} C_VEL
LIN {X 0,Y 404.097,Z 255.649,A -85,B 0,C 180,E1 -10763.131,E2 -10763.131} C_VEL
LIN {X 0,Y 404.109,Z 255.644,A -85,B 0,C 180,E1 -10766.194,E2 -10766.194} C_VEL
LIN {X 0,Y 404.113,Z 255.645,A -85,B 0,C 180,E1 -10769.721,E2 -10769.721} C_VEL
LIN {X 0,Y 404.166,Z 255.644,A -85,B 0,C 180,E1 -10773.129,E2 -10773.129} C_VEL
LIN {X 0,Y 404.146,Z 255.643,A -85,B 0,C 180,E1 -10775.34,E2 -10775.34} C_VEL
LIN {X 0,Y 404.113,Z 255.646,A -85,B 0,C 180,E1 -10778.587,E2 -10778.587} C_VEL
LIN {X 0,Y 404.182,Z 255.635,A -85,B 0,C 180,E1 -10781.768,E2 -10781.768} C_VEL
LIN {X 0,Y 404.184,Z 255.64,A -85,B 0,C 180,E1 -10784.888,E2 -10784.888} C_VEL
LIN {X 0,Y 404.238,Z 255.628,A -85,B 0,C 180,E1 -10787.965,E2 -10787.965} C_VEL
LIN {X 0,Y 404.251,Z 255.628,A -85,B 0,C 180,E1 -10791.005,E2 -10791.005} C_VEL
LIN {X 0,Y 404.383,Z 255.611,A -85,B 0,C 180,E1 -10794.021,E2 -10794.021} C_VEL
LIN {X 0,Y 404.468,Z 255.602,A -85,B 0,C 180,E1 -10798.014,E2 -10798.014} C_VEL
LIN {X 0,Y 404.393,Z 255.609,A -85,B 0,C 180,E1 -10801.002,E2 -10801.002} C_VEL
LIN {X 0,Y 404.381,Z 255.61,A -85,B 0,C 180,E1 -10802.994,E2 -10802.994} C_VEL
LIN {X 0,Y 404.337,Z 255.615,A -85,B 0,C 180,E1 -10806.994,E2 -10806.994} C_VEL
LIN {X 0,Y 404.252,Z 255.633,A -85,B 0,C 180,E1 -10810.017,E2 -10810.017} C_VEL
LIN {X 0,Y 404.268,Z 255.624,A -85,B 0,C 180,E1 -10813.216,E2 -10813.216} C_VEL
LIN {X 0,Y 404.179,Z 255.636,A -85,B 0,C 180,E1 -10817.199,E2 -10817.199} C_VEL
LIN {X 0,Y 404.159,Z 255.638,A -85,B 0,C 180,E1 -10820.357,E2 -10820.357} C_VEL
LIN {X 0,Y 404.153,Z 255.645,A -85,B 0,C 180,E1 -10823.58,E2 -10823.58} C_VEL
LIN {X 0,Y 404.109,Z 255.645,A -85,B 0,C 180,E1 -10826.888,E2 -10826.888} C_VEL
LIN {X 0,Y 404.15,Z 255.639,A -85,B 0,C 180,E1 -10830.289,E2 -10830.289} C_VEL
LIN {X 0,Y 404.146,Z 255.643,A -85,B 0,C 180,E1 -10833.817,E2 -10833.817} C_VEL
LIN {X 0,Y 404.142,Z 255.646,A -85,B 0,C 180,E1 -10836.877,E2 -10836.877} C_VEL
LIN {X 0,Y 404.143,Z 255.646,A -85,B 0,C 180,E1 -10838.763,E2 -10838.763} C_VEL
LIN {X 0,Y 404.242,Z 256.428,A -85,B 0,C 180,E1 -10840.097,E2 -10840.097} C_VEL
LIN {X 0,Y 404.698,Z 259.373,A -85,B 0,C 180,E1 -10843.167,E2 -10843.167} C_VEL
LIN {X 0,Y 405.106,Z 262.389,A -85,B 0,C 180,E1 -10846.058,E2 -10846.058} C_VEL
LIN {X 0,Y 405.273,Z 265.501,A -85,B 0,C 180,E1 -10848.779,E2 -10848.779} C_VEL
LIN {X 0,Y 405.093,Z 268.639,A -85,B 0,C 180,E1 -10851.35,E2 -10851.35} C_VEL
LIN {X 0,Y 404.608,Z 273.479,A -85,B 0,C 180,E1 -10855.027,E2 -10855.027} C_VEL
LIN {X 0,Y 404.2,Z 278.422,A -85,B 0,C 180,E1 -10858.56,E2 -10858.56} C_VEL
LIN {X 0,Y 403.85,Z 283.454,A -85,B 0,C 180,E1 -10861.975,E2 -10861.975} C_VEL
LIN {X 0,Y 403.547,Z 288.557,A -85,B 0,C 180,E1 -10865.294,E2 -10865.294} C_VEL
LIN {X 0,Y 403.294,Z 293.715,A -85,B 0,C 180,E1 -10868.534,E2 -10868.534} C_VEL
LIN {X 0,Y 403.091,Z 298.926,A -85,B 0,C 180,E1 -10871.71,E2 -10871.71} C_VEL
LIN {X 0,Y 403.103,Z 299.654,A -85,B 0,C 180,E1 -10872.123,E2 -10872.123} C_VEL
LIN {X 0,Y 405.07,Z 309.862,A -85,B 0,C 180,E1 -10872.525,E2 -10872.525} C_VEL
LIN {X 0,Y 406.795,Z 319.869,A -85,B 0,C 180,E1 -10873.034,E2 -10873.034} C_VEL
LIN {X 0,Y 407.952,Z 328.664,A -85,B 0,C 180,E1 -10873.573,E2 -10873.573} C_VEL
LIN {X 0,Y 407.331,Z 338.448,A -85,B 0,C 180,E1 -10874.232,E2 -10874.232} C_VEL
LIN {X 0,Y 406.668,Z 347.447,A -85,B 0,C 180,E1 -10874.976,E2 -10874.976} C_VEL
LIN {X 0,Y 406.048,Z 356.205,A -85,B 0,C 180,E1 -10875.852,E2 -10875.852} C_VEL
LIN {X 0,Y 405.531,Z 363.58,A -85,B 0,C 180,E1 -10876.725,E2 -10876.725} C_VEL
LIN {X 0,Y 404.961,Z 370.803,A -85,B 0,C 180,E1 -10877.726,E2 -10877.726} C_VEL
LIN {X 0,Y 404.439,Z 377.007,A -85,B 0,C 180,E1 -10878.727,E2 -10878.727} C_VEL
LIN {X 0,Y 403.912,Z 383.547,A -85,B 0,C 180,E1 -10879.98,E2 -10879.98} C_VEL
LIN {X 0,Y 403.605,Z 388.052,A -85,B 0,C 180,E1 -10880.984,E2 -10880.984} C_VEL
LIN {X 0,Y 403.225,Z 393.544,A -85,B 0,C 180,E1 -10882.489,E2 -10882.489} C_VEL
LIN {X 0,Y 403.004,Z 397.87,A -85,B 0,C 180,E1 -10883.994,E2 -10883.994} C_VEL
LIN {X 0,Y 402.962,Z 400.238,A -85,B 0,C 180,E1 -10884.997,E2 -10884.997} C_VEL
LIN {X 0,Y 402.868,Z 402.036,A -85,B 0,C 180,E1 -10885.999,E2 -10885.999} C_VEL
LIN {X 0,Y 402.868,Z 404.482,A -85,B 0,C 180,E1 -10888.001,E2 -10888.001} C_VEL
LIN {X 0,Y 402.854,Z 405.07,A -85,B 0,C 180,E1 -10889,E2 -10889} C_VEL
LIN {X 0,Y 402.854,Z 405.07,A -85,B 0,C 180,E1 -10891,E2 -10891} C_VEL
LIN {X 0,Y 402.868,Z 404.482,A -85,B 0,C 180,E1 -10891.999,E2 -10891.999} C_VEL
LIN {X 0,Y 402.868,Z 402.036,A -85,B 0,C 180,E1 -10894.001,E2 -10894.001} C_VEL
LIN {X 0,Y 402.967,Z 399.088,A -85,B 0,C 180,E1 -10895.504,E2 -10895.504} C_VEL
LIN {X 0,Y 403.131,Z 395.098,A -85,B 0,C 180,E1 -10897.009,E2 -10897.009} C_VEL
LIN {X 0,Y 403.444,Z 389.967,A -85,B 0,C 180,E1 -10898.515,E2 -10898.515} C_VEL
LIN {X 0,Y 403.836,Z 384.704,A -85,B 0,C 180,E1 -10899.769,E2 -10899.769} C_VEL
LIN {X 0,Y 404.277,Z 378.383,A -85,B 0,C 180,E1 -10901.024,E2 -10901.024} C_VEL
LIN {X 0,Y 404.82,Z 372.431,A -85,B 0,C 180,E1 -10902.024,E2 -10902.024} C_VEL
LIN {X 0,Y 405.374,Z 365.5,A -85,B 0,C 180,E1 -10903.025,E2 -10903.025} C_VEL
LIN {X 0,Y 405.979,Z 357.316,A -85,B 0,C 180,E1 -10904.025,E2 -10904.025} C_VEL
LIN {X 0,Y 406.568,Z 348.793,A -85,B 0,C 180,E1 -10904.9,E2 -10904.9} C_VEL
LIN {X 0,Y 407.227,Z 340.081,A -85,B 0,C 180,E1 -10905.644,E2 -10905.644} C_VEL
LIN {X 0,Y 407.938,Z 330.34,A -85,B 0,C 180,E1 -10906.32,E2 -10906.32} C_VEL
LIN {X 0,Y 407.368,Z 323.768,A -85,B 0,C 180,E1 -10906.747,E2 -10906.747} C_VEL
LIN {X 0,Y 405.428,Z 311.587,A -85,B 0,C 180,E1 -10907.395,E2 -10907.395} C_VEL
LIN {X 0,Y 403.256,Z 300.91,A -85,B 0,C 180,E1 -10907.839,E2 -10907.839} C_VEL
LIN {X 0,Y 403.096,Z 299.627,A -85,B 0,C 180,E1 -10907.893,E2 -10907.893} C_VEL
LIN {X 0,Y 403.246,Z 295.438,A -85,B 0,C 180,E1 -10910.4,E2 -10910.4} C_VEL
LIN {X 0,Y 403.434,Z 290.259,A -85,B 0,C 180,E1 -10913.62,E2 -10913.62} C_VEL
LIN {X 0,Y 403.75,Z 285.137,A -85,B 0,C 180,E1 -10916.909,E2 -10916.909} C_VEL
LIN {X 0,Y 404.059,Z 280.084,A -85,B 0,C 180,E1 -10920.292,E2 -10920.292} C_VEL
LIN {X 0,Y 404.447,Z 275.127,A -85,B 0,C 180,E1 -10923.783,E2 -10923.783} C_VEL
LIN {X 0,Y 404.854,Z 270.779,A -85,B 0,C 180,E1 -10927.005,E2 -10927.005} C_VEL
LIN {X 0,Y 405.196,Z 267.069,A -85,B 0,C 180,E1 -10929.922,E2 -10929.922} C_VEL
LIN {X 0,Y 405.293,Z 263.934,A -85,B 0,C 180,E1 -10932.553,E2 -10932.553} C_VEL
LIN {X 0,Y 404.932,Z 260.861,A -85,B 0,C 180,E1 -10935.364,E2 -10935.364} C_VEL
LIN {X 0,Y 404.427,Z 257.596,A -85,B 0,C 180,E1 -10938.669,E2 -10938.669} C_VEL
LIN {X 0,Y 404.241,Z 256.384,A -85,B 0,C 180,E1 -10939.959,E2 -10939.959} C_VEL
LIN {X 0,Y 404.148,Z 255.644,A -85,B 0,C 180,E1 -10941.492,E2 -10941.492} C_VEL
LIN {X 0,Y 404.182,Z 255.64,A -85,B 0,C 180,E1 -10944.979,E2 -10944.979} C_VEL
LIN {X 0,Y 404.145,Z 255.644,A -85,B 0,C 180,E1 -10948.439,E2 -10948.439} C_VEL
LIN {X 0,Y 404.156,Z 255.641,A -85,B 0,C 180,E1 -10950.858,E2 -10950.858} C_VEL
LIN {X 0,Y 404.158,Z 255.641,A -85,B 0,C 180,E1 -10954.719,E2 -10954.719} C_VEL
LIN {X 0,Y 404.17,Z 255.636,A -85,B 0,C 180,E1 -10957.503,E2 -10957.503} C_VEL
LIN {X 0,Y 404.16,Z 255.64,A -85,B 0,C 180,E1 -10960.702,E2 -10960.702} C_VEL
LIN {X 0,Y 404.181,Z 255.638,A -85,B 0,C 180,E1 -10963.841,E2 -10963.841} C_VEL
LIN {X 0,Y 404.284,Z 255.622,A -85,B 0,C 180,E1 -10966.934,E2 -10966.934} C_VEL
LIN {X 0,Y 404.252,Z 255.633,A -85,B 0,C 180,E1 -10969.983,E2 -10969.983} C_VEL
LIN {X 0,Y 404.337,Z 255.615,A -85,B 0,C 180,E1 -10973.006,E2 -10973.006} C_VEL
LIN {X 0,Y 404.252,Z 255.626,A -85,B 0,C 180,E1 -10975.008,E2 -10975.008} C_VEL
LIN {X 0,Y 404.463,Z 255.603,A -85,B 0,C 180,E1 -10978.003,E2 -10978.003} C_VEL
LIN {X 0,Y 404.339,Z 255.616,A -85,B 0,C 180,E1 -10980.99,E2 -10980.99} C_VEL
LIN {X 0,Y 404.395,Z 255.609,A -85,B 0,C 180,E1 -10982.983,E2 -10982.983} C_VEL
LIN {X 0,Y 404.37,Z 255.613,A -85,B 0,C 180,E1 -10986.982,E2 -10986.982} C_VEL
LIN {X 0,Y 404.234,Z 255.631,A -85,B 0,C 180,E1 -10991.019,E2 -10991.019} C_VEL
LIN {X 0,Y 404.19,Z 255.634,A -85,B 0,C 180,E1 -10994.082,E2 -10994.082} C_VEL
LIN {X 0,Y 404.181,Z 255.642,A -85,B 0,C 180,E1 -10997.186,E2 -10997.186} C_VEL
LIN {X 0,Y 404.14,Z 255.64,A -85,B 0,C 180,E1 -11000.345,E2 -11000.345} C_VEL
LIN {X 0,Y 404.136,Z 255.641,A -85,B 0,C 180,E1 -11003.569,E2 -11003.569} C_VEL
LIN {X 0,Y 404.155,Z 255.638,A -85,B 0,C 180,E1 -11005.76,E2 -11005.76} C_VEL
LIN {X 0,Y 404.165,Z 255.637,A -85,B 0,C 180,E1 -11007.994,E2 -11007.994} C_VEL
LIN {X 0,Y 404.105,Z 255.644,A -85,B 0,C 180,E1 -11011.552,E2 -11011.552} C_VEL
LIN {X 0,Y 404.148,Z 255.642,A -85,B 0,C 180,E1 -11015.01,E2 -11015.01} C_VEL
LIN {X 0,Y 404.108,Z 255.648,A -85,B 0,C 180,E1 -11018.752,E2 -11018.752} C_VEL
LIN {X 0,Y 404.145,Z 255.639,A -85,B 0,C 180,E1 -11021.604,E2 -11021.604} C_VEL
LIN {X 0,Y 404.152,Z 255.643,A -85,B 0,C 180,E1 -11024.524,E2 -11024.524} C_VEL
LIN {X 0,Y 404.163,Z 255.637,A -85,B 0,C 180,E1 -11027.3,E2 -11027.3} C_VEL
LIN {X 0,Y 404.12,Z 255.646,A -85,B 0,C 180,E1 -11029.95,E2 -11029.95} C_VEL
LIN {X 0,Y 404.089,Z 255.646,A -85,B 0,C 180,E1 -11033.12,E2 -11033.12} C_VEL
LIN {X 0,Y 404.091,Z 255.651,A -85,B 0,C 180,E1 -11036.183,E2 -11036.183} C_VEL
LIN {X 0,Y 404.099,Z 255.65,A -85,B 0,C 180,E1 -11039.712,E2 -11039.712} C_VEL
LIN {X 0,Y 404.138,Z 255.641,A -85,B 0,C 180,E1 -11043.119,E2 -11043.119} C_VEL
LIN {X 0,Y 404.126,Z 255.642,A -85,B 0,C 180,E1 -11046.423,E2 -11046.423} C_VEL
LIN {X 0,Y 404.166,Z 255.642,A -85,B 0,C 180,E1 -11049.858,E2 -11049.858} C_VEL
LIN {X 0,Y 404.157,Z 255.643,A -85,B 0,C 180,E1 -11052.989,E2 -11052.989} C_VEL
LIN {X 0,Y 404.204,Z 255.638,A -85,B 0,C 180,E1 -11056.787,E2 -11056.787} C_VEL
LIN {X 0,Y 404.212,Z 255.637,A -85,B 0,C 180,E1 -11059.987,E2 -11059.987} C_VEL
LIN {X 0,Y 404.38,Z 255.615,A -85,B 0,C 180,E1 -11063.012,E2 -11063.012} C_VEL
LIN {X 0,Y 404.229,Z 255.636,A -85,B 0,C 180,E1 -11065.013,E2 -11065.013} C_VEL
LIN {X 0,Y 404.419,Z 255.609,A -85,B 0,C 180,E1 -11068.008,E2 -11068.008} C_VEL
LIN {X 0,Y 404.548,Z 255.595,A -85,B 0,C 180,E1 -11070,E2 -11070} C_VEL
LIN {X 0,Y 404.367,Z 255.616,A -85,B 0,C 180,E1 -11072.989,E2 -11072.989} C_VEL
LIN {X 0,Y 404.38,Z 255.615,A -85,B 0,C 180,E1 -11076.988,E2 -11076.988} C_VEL
LIN {X 0,Y 404.212,Z 255.637,A -85,B 0,C 180,E1 -11080.013,E2 -11080.013} C_VEL
LIN {X 0,Y 404.204,Z 255.638,A -85,B 0,C 180,E1 -11083.213,E2 -11083.213} C_VEL
LIN {X 0,Y 404.157,Z 255.643,A -85,B 0,C 180,E1 -11087.011,E2 -11087.011} C_VEL
LIN {X 0,Y 404.147,Z 255.646,A -85,B 0,C 180,E1 -11090.352,E2 -11090.352} C_VEL
LIN {X 0,Y 404.135,Z 255.64,A -85,B 0,C 180,E1 -11091.884,E2 -11091.884} C_VEL
LIN {X 0,Y 403.483,Z 255.728,A -85,B 0,C 180,E1 -11092.716,E2 -11092.716} C_VEL
LIN {X 0,Y 400.63,Z 256.091,A -85,B 0,C 180,E1 -11094.066,E2 -11094.066} C_VEL
LIN {X 0,Y 398.205,Z 256.394,A -85,B 0,C 180,E1 -11095.158,E2 -11095.158} C_VEL
LIN {X 0,Y 397.163,Z 256.518,A -85,B 0,C 180,E1 -11096.002,E2 -11096.002} C_VEL
LIN {X 0,Y 397.078,Z 256.526,A -85,B 0,C 180,E1 -11096.287,E2 -11096.287} C_VEL
LIN {X 0,Y 397.07,Z 256.523,A -85,B 0,C 180,E1 -11098.547,E2 -11098.547} C_VEL
LIN {X 0,Y 397.057,Z 256.529,A -85,B 0,C 180,E1 -11102.073,E2 -11102.073} C_VEL
LIN {X 0,Y 397.067,Z 256.523,A -85,B 0,C 180,E1 -11105.508,E2 -11105.508} C_VEL
LIN {X 0,Y 397.087,Z 256.518,A -85,B 0,C 180,E1 -11108.867,E2 -11108.867} C_VEL
LIN {X 0,Y 397.113,Z 256.517,A -85,B 0,C 180,E1 -11112.26,E2 -11112.26} C_VEL
LIN {X 0,Y 397.105,Z 256.517,A -85,B 0,C 180,E1 -11115.065,E2 -11115.065} C_VEL
LIN {X 0,Y 397.111,Z 256.518,A -85,B 0,C 180,E1 -11118.013,E2 -11118.013} C_VEL
LIN {X 0,Y 397.058,Z 256.526,A -85,B 0,C 180,E1 -11121.73,E2 -11121.73} C_VEL
LIN {X 0,Y 397.089,Z 256.523,A -85,B 0,C 180,E1 -11125.513,E2 -11125.513} C_VEL
LIN {X 0,Y 397.045,Z 256.529,A -85,B 0,C 180,E1 -11129.124,E2 -11129.124} C_VEL
LIN {X 0,Y 397.164,Z 256.51,A -85,B 0,C 180,E1 -11132.616,E2 -11132.616} C_VEL
LIN {X 0,Y 397.101,Z 256.517,A -85,B 0,C 180,E1 -11135.988,E2 -11135.988} C_VEL
LIN {X 0,Y 397.115,Z 256.515,A -85,B 0,C 180,E1 -11139.711,E2 -11139.711} C_VEL
LIN {X 0,Y 397.161,Z 256.516,A -85,B 0,C 180,E1 -11142.851,E2 -11142.851} C_VEL
LIN {X 0,Y 397.212,Z 256.51,A -85,B 0,C 180,E1 -11146.709,E2 -11146.709} C_VEL
LIN {X 0,Y 397.2,Z 256.505,A -85,B 0,C 180,E1 -11149.815,E2 -11149.815} C_VEL
LIN {X 0,Y 397.318,Z 256.492,A -85,B 0,C 180,E1 -11152.894,E2 -11152.894} C_VEL
LIN {X 0,Y 397.231,Z 256.502,A -85,B 0,C 180,E1 -11154.931,E2 -11154.931} C_VEL
LIN {X 0,Y 397.437,Z 256.477,A -85,B 0,C 180,E1 -11157.979,E2 -11157.979} C_VEL
LIN {X 0,Y 397.432,Z 256.48,A -85,B 0,C 180,E1 -11162.033,E2 -11162.033} C_VEL
LIN {X 0,Y 397.316,Z 256.496,A -85,B 0,C 180,E1 -11166.098,E2 -11166.098} C_VEL
LIN {X 0,Y 397.232,Z 256.5,A -85,B 0,C 180,E1 -11169.168,E2 -11169.168} C_VEL
LIN {X 0,Y 397.218,Z 256.505,A -85,B 0,C 180,E1 -11172.263,E2 -11172.263} C_VEL
LIN {X 0,Y 397.125,Z 256.516,A -85,B 0,C 180,E1 -11175.399,E2 -11175.399} C_VEL
LIN {X 0,Y 397.113,Z 256.515,A -85,B 0,C 180,E1 -11178.581,E2 -11178.581} C_VEL
LIN {X 0,Y 397.098,Z 256.522,A -85,B 0,C 180,E1 -11181.823,E2 -11181.823} C_VEL
LIN {X 0,Y 397.108,Z 256.518,A -85,B 0,C 180,E1 -11185.14,E2 -11185.14} C_VEL
LIN {X 0,Y 397.07,Z 256.521,A -85,B 0,C 180,E1 -11188.553,E2 -11188.553} C_VEL
LIN {X 0,Y 397.088,Z 256.52,A -85,B 0,C 180,E1 -11191.839,E2 -11191.839} C_VEL
LIN {X 0,Y 397.126,Z 256.518,A -85,B 0,C 180,E1 -11194.498,E2 -11194.498} C_VEL
LIN {X 0,Y 397.101,Z 256.523,A -85,B 0,C 180,E1 -11198.28,E2 -11198.28} C_VEL
LIN {X 0,Y 397.105,Z 256.522,A -85,B 0,C 180,E1 -11198.858,E2 -11198.858} C_VEL
LIN {X 0,Y 397.534,Z 259.597,A -85,B 0,C 180,E1 -11202.211,E2 -11202.211} C_VEL
LIN {X 0,Y 397.954,Z 262.435,A -85,B 0,C 180,E1 -11205.057,E2 -11205.057} C_VEL
LIN {X 0,Y 398.264,Z 265.509,A -85,B 0,C 180,E1 -11207.89,E2 -11207.89} C_VEL
LIN {X 0,Y 398.063,Z 269.168,A -85,B 0,C 180,E1 -11210.977,E2 -11210.977} C_VEL
LIN {X 0,Y 397.79,Z 271.823,A -85,B 0,C 180,E1 -11213.081,E2 -11213.081} C_VEL
LIN {X 0,Y 397.318,Z 276.711,A -85,B 0,C 180,E1 -11216.747,E2 -11216.747} C_VEL
LIN {X 0,Y 396.955,Z 281.676,A -85,B 0,C 180,E1 -11220.282,E2 -11220.282} C_VEL
LIN {X 0,Y 396.617,Z 286.739,A -85,B 0,C 180,E1 -11223.705,E2 -11223.705} C_VEL
LIN {X 0,Y 396.308,Z 292.192,A -85,B 0,C 180,E1 -11227.249,E2 -11227.249} C_VEL
LIN {X 0,Y 396.156,Z 297.001,A -85,B 0,C 180,E1 -11230.302,E2 -11230.302} C_VEL
LIN {X 0,Y 396.007,Z 299.484,A -85,B 0,C 180,E1 -11231.793,E2 -11231.793} C_VEL
LIN {X 0,Y 398.093,Z 309.865,A -85,B 0,C 180,E1 -11232.217,E2 -11232.217} C_VEL
LIN {X 0,Y 399.845,Z 320.113,A -85,B 0,C 180,E1 -11232.754,E2 -11232.754} C_VEL
LIN {X 0,Y 401.046,Z 328.851,A -85,B 0,C 180,E1 -11233.308,E2 -11233.308} C_VEL
LIN {X 0,Y 400.633,Z 336.605,A -85,B 0,C 180,E1 -11233.831,E2 -11233.831} C_VEL
LIN {X 0,Y 399.925,Z 345.883,A -85,B 0,C 180,E1 -11234.586,E2 -11234.586} C_VEL
LIN {X 0,Y 399.224,Z 354.837,A -85,B 0,C 180,E1 -11235.472,E2 -11235.472} C_VEL
LIN {X 0,Y 398.571,Z 363.367,A -85,B 0,C 180,E1 -11236.489,E2 -11236.489} C_VEL
LIN {X 0,Y 397.984,Z 370.591,A -85,B 0,C 180,E1 -11237.507,E2 -11237.507} C_VEL
LIN {X 0,Y 397.446,Z 376.795,A -85,B 0,C 180,E1 -11238.526,E2 -11238.526} C_VEL
LIN {X 0,Y 396.907,Z 383.335,A -85,B 0,C 180,E1 -11239.801,E2 -11239.801} C_VEL
LIN {X 0,Y 396.566,Z 387.839,A -85,B 0,C 180,E1 -11240.822,E2 -11240.822} C_VEL
LIN {X 0,Y 396.175,Z 393.333,A -85,B 0,C 180,E1 -11242.354,E2 -11242.354} C_VEL
LIN {X 0,Y 395.925,Z 397.658,A -85,B 0,C 180,E1 -11243.886,E2 -11243.886} C_VEL
LIN {X 0,Y 395.878,Z 400.027,A -85,B 0,C 180,E1 -11244.908,E2 -11244.908} C_VEL
LIN {X 0,Y 395.792,Z 401.825,A -85,B 0,C 180,E1 -11245.927,E2 -11245.927} C_VEL
LIN {X 0,Y 395.766,Z 404.271,A -85,B 0,C 180,E1 -11247.965,E2 -11247.965} C_VEL
LIN {X 0,Y 395.784,Z 404.86,A -85,B 0,C 180,E1 -11248.983,E2 -11248.983} C_VEL
LIN {X 0,Y 395.784,Z 404.86,A -85,B 0,C 180,E1 -11251.017,E2 -11251.017} C_VEL
LIN {X 0,Y 395.766,Z 404.271,A -85,B 0,C 180,E1 -11252.035,E2 -11252.035} C_VEL
LIN {X 0,Y 395.792,Z 401.825,A -85,B 0,C 180,E1 -11254.073,E2 -11254.073} C_VEL
LIN {X 0,Y 395.872,Z 398.875,A -85,B 0,C 180,E1 -11255.603,E2 -11255.603} C_VEL
LIN {X 0,Y 396.077,Z 394.887,A -85,B 0,C 180,E1 -11257.135,E2 -11257.135} C_VEL
LIN {X 0,Y 396.4,Z 389.755,A -85,B 0,C 180,E1 -11258.667,E2 -11258.667} C_VEL
LIN {X 0,Y 396.802,Z 384.491,A -85,B 0,C 180,E1 -11259.944,E2 -11259.944} C_VEL
LIN {X 0,Y 397.278,Z 378.17,A -85,B 0,C 180,E1 -11261.221,E2 -11261.221} C_VEL
LIN {X 0,Y 397.834,Z 372.218,A -85,B 0,C 180,E1 -11262.239,E2 -11262.239} C_VEL
LIN {X 0,Y 398.424,Z 365.288,A -85,B 0,C 180,E1 -11263.256,E2 -11263.256} C_VEL
LIN {X 0,Y 399.054,Z 357.103,A -85,B 0,C 180,E1 -11264.274,E2 -11264.274} C_VEL
LIN {X 0,Y 399.691,Z 348.723,A -85,B 0,C 180,E1 -11265.149,E2 -11265.149} C_VEL
LIN {X 0,Y 400.363,Z 339.868,A -85,B 0,C 180,E1 -11265.919,E2 -11265.919} C_VEL
LIN {X 0,Y 401.078,Z 330.421,A -85,B 0,C 180,E1 -11266.589,E2 -11266.589} C_VEL
LIN {X 0,Y 400.095,Z 321.898,A -85,B 0,C 180,E1 -11267.144,E2 -11267.144} C_VEL
LIN {X 0,Y 398.321,Z 311.184,A -85,B 0,C 180,E1 -11267.722,E2 -11267.722} C_VEL
LIN {X 0,Y 396.081,Z 300.266,A -85,B 0,C 180,E1 -11268.184,E2 -11268.184} C_VEL
LIN {X 0,Y 396.03,Z 299.442,A -85,B 0,C 180,E1 -11268.223,E2 -11268.223} C_VEL
LIN {X 0,Y 396.164,Z 295.267,A -85,B 0,C 180,E1 -11270.781,E2 -11270.781} C_VEL
LIN {X 0,Y 396.4,Z 290.105,A -85,B 0,C 180,E1 -11274.065,E2 -11274.065} C_VEL
LIN {X 0,Y 396.771,Z 284.673,A -85,B 0,C 180,E1 -11277.663,E2 -11277.663} C_VEL
LIN {X 0,Y 397.066,Z 280.014,A -85,B 0,C 180,E1 -11280.883,E2 -11280.883} C_VEL
LIN {X 0,Y 397.469,Z 275.069,A -85,B 0,C 180,E1 -11284.459,E2 -11284.459} C_VEL
LIN {X 0,Y 397.868,Z 271.264,A -85,B 0,C 180,E1 -11287.35,E2 -11287.35} C_VEL
LIN {X 0,Y 398.19,Z 267.236,A -85,B 0,C 180,E1 -11290.624,E2 -11290.624} C_VEL
LIN {X 0,Y 398.279,Z 265.441,A -85,B 0,C 180,E1 -11292.167,E2 -11292.167} C_VEL
LIN {X 0,Y 397.963,Z 262.299,A -85,B 0,C 180,E1 -11295.053,E2 -11295.053} C_VEL
LIN {X 0,Y 397.501,Z 259.424,A -85,B 0,C 180,E1 -11297.95,E2 -11297.95} C_VEL
LIN {X 0,Y 397.105,Z 256.522,A -85,B 0,C 180,E1 -11301.142,E2 -11301.142} C_VEL
LIN {X 0,Y 397.108,Z 256.52,A -85,B 0,C 180,E1 -11304.498,E2 -11304.498} C_VEL
LIN {X 0,Y 397.084,Z 256.519,A -85,B 0,C 180,E1 -11307.924,E2 -11307.924} C_VEL
LIN {X 0,Y 397.123,Z 256.518,A -85,B 0,C 180,E1 -11310.291,E2 -11310.291} C_VEL
LIN {X 0,Y 397.081,Z 256.52,A -85,B 0,C 180,E1 -11313.733,E2 -11313.733} C_VEL
LIN {X 0,Y 397.105,Z 256.517,A -85,B 0,C 180,E1 -11317.081,E2 -11317.081} C_VEL
LIN {X 0,Y 397.133,Z 256.519,A -85,B 0,C 180,E1 -11320.347,E2 -11320.347} C_VEL
LIN {X 0,Y 397.129,Z 256.514,A -85,B 0,C 180,E1 -11323.546,E2 -11323.546} C_VEL
LIN {X 0,Y 397.231,Z 256.502,A -85,B 0,C 180,E1 -11326.698,E2 -11326.698} C_VEL
LIN {X 0,Y 397.213,Z 256.507,A -85,B 0,C 180,E1 -11329.803,E2 -11329.803} C_VEL
LIN {X 0,Y 397.289,Z 256.493,A -85,B 0,C 180,E1 -11332.881,E2 -11332.881} C_VEL
LIN {X 0,Y 397.223,Z 256.501,A -85,B 0,C 180,E1 -11334.919,E2 -11334.919} C_VEL
LIN {X 0,Y 397.432,Z 256.48,A -85,B 0,C 180,E1 -11337.967,E2 -11337.967} C_VEL
LIN {X 0,Y 397.437,Z 256.477,A -85,B 0,C 180,E1 -11342.021,E2 -11342.021} C_VEL
LIN {X 0,Y 397.311,Z 256.49,A -85,B 0,C 180,E1 -11346.583,E2 -11346.583} C_VEL
LIN {X 0,Y 397.221,Z 256.506,A -85,B 0,C 180,E1 -11349.156,E2 -11349.156} C_VEL
LIN {X 0,Y 397.202,Z 256.504,A -85,B 0,C 180,E1 -11352.252,E2 -11352.252} C_VEL
LIN {X 0,Y 397.157,Z 256.515,A -85,B 0,C 180,E1 -11355.386,E2 -11355.386} C_VEL
LIN {X 0,Y 397.135,Z 256.514,A -85,B 0,C 180,E1 -11358.567,E2 -11358.567} C_VEL
LIN {X 0,Y 397.07,Z 256.521,A -85,B 0,C 180,E1 -11361.812,E2 -11361.812} C_VEL
LIN {X 0,Y 397.124,Z 256.515,A -85,B 0,C 180,E1 -11365.506,E2 -11365.506} C_VEL
LIN {X 0,Y 397.091,Z 256.521,A -85,B 0,C 180,E1 -11368.537,E2 -11368.537} C_VEL
LIN {X 0,Y 397.043,Z 256.525,A -85,B 0,C 180,E1 -11372.066,E2 -11372.066} C_VEL
LIN {X 0,Y 397.082,Z 256.519,A -85,B 0,C 180,E1 -11375.497,E2 -11375.497} C_VEL
LIN {X 0,Y 397.085,Z 256.522,A -85,B 0,C 180,E1 -11378.855,E2 -11378.855} C_VEL
LIN {X 0,Y 397.114,Z 256.52,A -85,B 0,C 180,E1 -11382.25,E2 -11382.25} C_VEL
LIN {X 0,Y 397.106,Z 256.517,A -85,B 0,C 180,E1 -11385.054,E2 -11385.054} C_VEL
LIN {X 0,Y 397.109,Z 256.52,A -85,B 0,C 180,E1 -11388.002,E2 -11388.002} C_VEL
LIN {X 0,Y 397.059,Z 256.524,A -85,B 0,C 180,E1 -11391.721,E2 -11391.721} C_VEL
LIN {X 0,Y 397.072,Z 256.522,A -85,B 0,C 180,E1 -11395.502,E2 -11395.502} C_VEL
LIN {X 0,Y 397.031,Z 256.526,A -85,B 0,C 180,E1 -11399.114,E2 -11399.114} C_VEL
LIN {X 0,Y 397.138,Z 256.512,A -85,B 0,C 180,E1 -11402.606,E2 -11402.606} C_VEL
LIN {X 0,Y 397.083,Z 256.523,A -85,B 0,C 180,E1 -11405.979,E2 -11405.979} C_VEL
LIN {X 0,Y 397.098,Z 256.52,A -85,B 0,C 180,E1 -11409.27,E2 -11409.27} C_VEL
LIN {X 0,Y 397.122,Z 256.519,A -85,B 0,C 180,E1 -11412.842,E2 -11412.842} C_VEL
LIN {X 0,Y 397.123,Z 256.519,A -85,B 0,C 180,E1 -11415.655,E2 -11415.655} C_VEL
LIN {X 0,Y 397.149,Z 256.516,A -85,B 0,C 180,E1 -11418.776,E2 -11418.776} C_VEL
LIN {X 0,Y 397.335,Z 256.492,A -85,B 0,C 180,E1 -11422.036,E2 -11422.036} C_VEL
LIN {X 0,Y 397.335,Z 256.493,A -85,B 0,C 180,E1 -11423.908,E2 -11423.908} C_VEL
LIN {X 0,Y 397.388,Z 256.485,A -85,B 0,C 180,E1 -11427.973,E2 -11427.973} C_VEL
LIN {X 0,Y 397.518,Z 256.471,A -85,B 0,C 180,E1 -11430,E2 -11430} C_VEL
LIN {X 0,Y 397.325,Z 256.493,A -85,B 0,C 180,E1 -11433.042,E2 -11433.042} C_VEL
LIN {X 0,Y 397.328,Z 256.493,A -85,B 0,C 180,E1 -11437.112,E2 -11437.112} C_VEL
LIN {X 0,Y 397.169,Z 256.514,A -85,B 0,C 180,E1 -11440.192,E2 -11440.192} C_VEL
LIN {X 0,Y 397.164,Z 256.514,A -85,B 0,C 180,E1 -11443.323,E2 -11443.323} C_VEL
LIN {X 0,Y 397.11,Z 256.522,A -85,B 0,C 180,E1 -11446.449,E2 -11446.449} C_VEL
LIN {X 0,Y 397.114,Z 256.516,A -85,B 0,C 180,E1 -11449.649,E2 -11449.649} C_VEL
LIN {X 0,Y 397.117,Z 256.515,A -85,B 0,C 180,E1 -11453.057,E2 -11453.057} C_VEL
LIN {X 0,Y 397.078,Z 256.526,A -85,B 0,C 180,E1 -11456.287,E2 -11456.287} C_VEL
LIN {X 0,Y 396.405,Z 256.604,A -85,B 0,C 180,E1 -11457.134,E2 -11457.134} C_VEL
LIN {X 0,Y 393.532,Z 256.964,A -85,B 0,C 180,E1 -11458.51,E2 -11458.51} C_VEL
LIN {X 0,Y 391.1,Z 257.268,A -85,B 0,C 180,E1 -11459.622,E2 -11459.622} C_VEL
LIN {X 0,Y 390.056,Z 257.398,A -85,B 0,C 180,E1 -11460.482,E2 -11460.482} C_VEL
LIN {X 0,Y 389.97,Z 257.406,A -85,B 0,C 180,E1 -11460.774,E2 -11460.774} C_VEL
LIN {X 0,Y 390.016,Z 257.406,A -85,B 0,C 180,E1 -11464.029,E2 -11464.029} C_VEL
LIN {X 0,Y 389.996,Z 257.405,A -85,B 0,C 180,E1 -11467.556,E2 -11467.556} C_VEL
LIN {X 0,Y 390.034,Z 257.397,A -85,B 0,C 180,E1 -11470.831,E2 -11470.831} C_VEL
LIN {X 0,Y 390.083,Z 257.395,A -85,B 0,C 180,E1 -11473.903,E2 -11473.903} C_VEL
LIN {X 0,Y 390.07,Z 257.393,A -85,B 0,C 180,E1 -11476.803,E2 -11476.803} C_VEL
LIN {X 0,Y 390.026,Z 257.404,A -85,B 0,C 180,E1 -11479.568,E2 -11479.568} C_VEL
LIN {X 0,Y 390.002,Z 257.401,A -85,B 0,C 180,E1 -11482.456,E2 -11482.456} C_VEL
LIN {X 0,Y 390.033,Z 257.398,A -85,B 0,C 180,E1 -11485.982,E2 -11485.982} C_VEL
LIN {X 0,Y 390.014,Z 257.4,A -85,B 0,C 180,E1 -11489.875,E2 -11489.875} C_VEL
LIN {X 0,Y 390.084,Z 257.396,A -85,B 0,C 180,E1 -11493.238,E2 -11493.238} C_VEL
LIN {X 0,Y 390.05,Z 257.399,A -85,B 0,C 180,E1 -11496.767,E2 -11496.767} C_VEL
LIN {X 0,Y 390.08,Z 257.391,A -85,B 0,C 180,E1 -11499.989,E2 -11499.989} C_VEL
LIN {X 0,Y 390.117,Z 257.389,A -85,B 0,C 180,E1 -11503.255,E2 -11503.255} C_VEL
LIN {X 0,Y 390.178,Z 257.384,A -85,B 0,C 180,E1 -11506.568,E2 -11506.568} C_VEL
LIN {X 0,Y 390.151,Z 257.382,A -85,B 0,C 180,E1 -11509.629,E2 -11509.629} C_VEL
LIN {X 0,Y 390.267,Z 257.372,A -85,B 0,C 180,E1 -11512.765,E2 -11512.765} C_VEL
LIN {X 0,Y 390.203,Z 257.379,A -85,B 0,C 180,E1 -11514.84,E2 -11514.84} C_VEL
LIN {X 0,Y 390.404,Z 257.353,A -85,B 0,C 180,E1 -11517.943,E2 -11517.943} C_VEL
LIN {X 0,Y 390.4,Z 257.356,A -85,B 0,C 180,E1 -11522.069,E2 -11522.069} C_VEL
LIN {X 0,Y 390.272,Z 257.373,A -85,B 0,C 180,E1 -11526.208,E2 -11526.208} C_VEL
LIN {X 0,Y 390.19,Z 257.378,A -85,B 0,C 180,E1 -11529.335,E2 -11529.335} C_VEL
LIN {X 0,Y 390.171,Z 257.381,A -85,B 0,C 180,E1 -11532.488,E2 -11532.488} C_VEL
LIN {X 0,Y 390.068,Z 257.398,A -85,B 0,C 180,E1 -11535.685,E2 -11535.685} C_VEL
LIN {X 0,Y 390.071,Z 257.393,A -85,B 0,C 180,E1 -11538.929,E2 -11538.929} C_VEL
LIN {X 0,Y 390.039,Z 257.398,A -85,B 0,C 180,E1 -11542.239,E2 -11542.239} C_VEL
LIN {X 0,Y 390.057,Z 257.399,A -85,B 0,C 180,E1 -11545.726,E2 -11545.726} C_VEL
LIN {X 0,Y 390.031,Z 257.4,A -85,B 0,C 180,E1 -11549.117,E2 -11549.117} C_VEL
LIN {X 0,Y 390.049,Z 257.396,A -85,B 0,C 180,E1 -11552.726,E2 -11552.726} C_VEL
LIN {X 0,Y 390.052,Z 257.399,A -85,B 0,C 180,E1 -11555.826,E2 -11555.826} C_VEL
LIN {X 0,Y 390.047,Z 257.401,A -85,B 0,C 180,E1 -11557.784,E2 -11557.784} C_VEL
LIN {X 0,Y 390.147,Z 258.033,A -85,B 0,C 180,E1 -11559.233,E2 -11559.233} C_VEL
LIN {X 0,Y 390.548,Z 260.968,A -85,B 0,C 180,E1 -11562.457,E2 -11562.457} C_VEL
LIN {X 0,Y 390.974,Z 263.976,A -85,B 0,C 180,E1 -11565.49,E2 -11565.49} C_VEL
LIN {X 0,Y 391.208,Z 267.054,A -85,B 0,C 180,E1 -11568.342,E2 -11568.342} C_VEL
LIN {X 0,Y 391.019,Z 270.217,A -85,B 0,C 180,E1 -11571.019,E2 -11571.019} C_VEL
LIN {X 0,Y 390.606,Z 274.014,A -85,B 0,C 180,E1 -11574.069,E2 -11574.069} C_VEL
LIN {X 0,Y 390.184,Z 278.278,A -85,B 0,C 180,E1 -11577.293,E2 -11577.293} C_VEL
LIN {X 0,Y 389.822,Z 283.249,A -85,B 0,C 180,E1 -11580.872,E2 -11580.872} C_VEL
LIN {X 0,Y 389.464,Z 288.485,A -85,B 0,C 180,E1 -11584.464,E2 -11584.464} C_VEL
LIN {X 0,Y 389.202,Z 293.396,A -85,B 0,C 180,E1 -11587.716,E2 -11587.716} C_VEL
LIN {X 0,Y 388.991,Z 298.554,A -85,B 0,C 180,E1 -11591.022,E2 -11591.022} C_VEL
LIN {X 0,Y 388.941,Z 299.351,A -85,B 0,C 180,E1 -11591.453,E2 -11591.453} C_VEL
LIN {X 0,Y 391.012,Z 309.412,A -85,B 0,C 180,E1 -11591.875,E2 -11591.875} C_VEL
LIN {X 0,Y 392.576,Z 318.524,A -85,B 0,C 180,E1 -11592.353,E2 -11592.353} C_VEL
LIN {X 0,Y 393.908,Z 327.503,A -85,B 0,C 180,E1 -11592.922,E2 -11592.922} C_VEL
LIN {X 0,Y 394.09,Z 333.444,A -85,B 0,C 180,E1 -11593.323,E2 -11593.323} C_VEL
LIN {X 0,Y 393.057,Z 345.671,A -85,B 0,C 180,E1 -11594.31,E2 -11594.31} C_VEL
LIN {X 0,Y 392.31,Z 354.624,A -85,B 0,C 180,E1 -11595.211,E2 -11595.211} C_VEL
LIN {X 0,Y 391.779,Z 361.573,A -85,B 0,C 180,E1 -11596.032,E2 -11596.032} C_VEL
LIN {X 0,Y 391.031,Z 370.379,A -85,B 0,C 180,E1 -11597.281,E2 -11597.281} C_VEL
LIN {X 0,Y 390.431,Z 376.582,A -85,B 0,C 180,E1 -11598.317,E2 -11598.317} C_VEL
LIN {X 0,Y 389.891,Z 383.123,A -85,B 0,C 180,E1 -11599.616,E2 -11599.616} C_VEL
LIN {X 0,Y 389.501,Z 387.626,A -85,B 0,C 180,E1 -11600.654,E2 -11600.654} C_VEL
LIN {X 0,Y 389.106,Z 393.12,A -85,B 0,C 180,E1 -11602.215,E2 -11602.215} C_VEL
LIN {X 0,Y 388.85,Z 397.446,A -85,B 0,C 180,E1 -11603.775,E2 -11603.775} C_VEL
LIN {X 0,Y 388.776,Z 399.815,A -85,B 0,C 180,E1 -11604.814,E2 -11604.814} C_VEL
LIN {X 0,Y 388.717,Z 401.614,A -85,B 0,C 180,E1 -11605.853,E2 -11605.853} C_VEL
LIN {X 0,Y 388.665,Z 404.059,A -85,B 0,C 180,E1 -11607.927,E2 -11607.927} C_VEL
LIN {X 0,Y 388.697,Z 404.649,A -85,B 0,C 180,E1 -11608.964,E2 -11608.964} C_VEL
LIN {X 0,Y 388.697,Z 404.649,A -85,B 0,C 180,E1 -11611.036,E2 -11611.036} C_VEL
LIN {X 0,Y 388.665,Z 404.059,A -85,B 0,C 180,E1 -11612.073,E2 -11612.073} C_VEL
LIN {X 0,Y 388.717,Z 401.614,A -85,B 0,C 180,E1 -11614.147,E2 -11614.147} C_VEL
LIN {X 0,Y 388.791,Z 398.384,A -85,B 0,C 180,E1 -11615.825,E2 -11615.825} C_VEL
LIN {X 0,Y 388.998,Z 394.674,A -85,B 0,C 180,E1 -11617.265,E2 -11617.265} C_VEL
LIN {X 0,Y 389.37,Z 389.544,A -85,B 0,C 180,E1 -11618.825,E2 -11618.825} C_VEL
LIN {X 0,Y 389.772,Z 384.279,A -85,B 0,C 180,E1 -11620.125,E2 -11620.125} C_VEL
LIN {X 0,Y 390.287,Z 377.958,A -85,B 0,C 180,E1 -11621.424,E2 -11621.424} C_VEL
LIN {X 0,Y 390.854,Z 372.005,A -85,B 0,C 180,E1 -11622.461,E2 -11622.461} C_VEL
LIN {X 0,Y 391.474,Z 365.075,A -85,B 0,C 180,E1 -11623.496,E2 -11623.496} C_VEL
LIN {X 0,Y 392.142,Z 356.891,A -85,B 0,C 180,E1 -11624.531,E2 -11624.531} C_VEL
LIN {X 0,Y 392.81,Z 348.51,A -85,B 0,C 180,E1 -11625.421,E2 -11625.421} C_VEL
LIN {X 0,Y 393.537,Z 339.657,A -85,B 0,C 180,E1 -11626.203,E2 -11626.203} C_VEL
LIN {X 0,Y 394.218,Z 330.482,A -85,B 0,C 180,E1 -11626.868,E2 -11626.868} C_VEL
LIN {X 0,Y 393.03,Z 321.256,A -85,B 0,C 180,E1 -11627.484,E2 -11627.484} C_VEL
LIN {X 0,Y 391.274,Z 310.856,A -85,B 0,C 180,E1 -11628.057,E2 -11628.057} C_VEL
LIN {X 0,Y 389.011,Z 300.044,A -85,B 0,C 180,E1 -11628.526,E2 -11628.526} C_VEL
LIN {X 0,Y 388.939,Z 299.255,A -85,B 0,C 180,E1 -11628.567,E2 -11628.567} C_VEL
LIN {X 0,Y 389.118,Z 295.078,A -85,B 0,C 180,E1 -11631.175,E2 -11631.175} C_VEL
LIN {X 0,Y 389.347,Z 289.974,A -85,B 0,C 180,E1 -11634.529,E2 -11634.529} C_VEL
LIN {X 0,Y 389.713,Z 284.924,A -85,B 0,C 180,E1 -11637.961,E2 -11637.961} C_VEL
LIN {X 0,Y 390.062,Z 279.934,A -85,B 0,C 180,E1 -11641.5,E2 -11641.5} C_VEL
LIN {X 0,Y 390.528,Z 275.011,A -85,B 0,C 180,E1 -11645.16,E2 -11645.16} C_VEL
LIN {X 0,Y 390.866,Z 271.789,A -85,B 0,C 180,E1 -11647.702,E2 -11647.702} C_VEL
LIN {X 0,Y 391.125,Z 268.624,A -85,B 0,C 180,E1 -11650.305,E2 -11650.305} C_VEL
LIN {X 0,Y 391.188,Z 265.498,A -85,B 0,C 180,E1 -11653.054,E2 -11653.054} C_VEL
LIN {X 0,Y 390.792,Z 262.448,A -85,B 0,C 180,E1 -11656,E2 -11656} C_VEL
LIN {X 0,Y 390.29,Z 259.071,A -85,B 0,C 180,E1 -11659.585,E2 -11659.585} C_VEL
LIN {X 0,Y 390.116,Z 257.916,A -85,B 0,C 180,E1 -11660.906,E2 -11660.906} C_VEL
LIN {X 0,Y 390.048,Z 257.401,A -85,B 0,C 180,E1 -11662.447,E2 -11662.447} C_VEL
LIN {X 0,Y 390.071,Z 257.395,A -85,B 0,C 180,E1 -11666.041,E2 -11666.041} C_VEL
LIN {X 0,Y 390.05,Z 257.395,A -85,B 0,C 180,E1 -11669.866,E2 -11669.866} C_VEL
LIN {X 0,Y 390.036,Z 257.397,A -85,B 0,C 180,E1 -11673.221,E2 -11673.221} C_VEL
LIN {X 0,Y 390.065,Z 257.396,A -85,B 0,C 180,E1 -11676.762,E2 -11676.762} C_VEL
LIN {X 0,Y 390.089,Z 257.394,A -85,B 0,C 180,E1 -11679.977,E2 -11679.977} C_VEL
LIN {X 0,Y 390.108,Z 257.388,A -85,B 0,C 180,E1 -11683.242,E2 -11683.242} C_VEL
LIN {X 0,Y 390.196,Z 257.379,A -85,B 0,C 180,E1 -11686.556,E2 -11686.556} C_VEL
LIN {X 0,Y 390.164,Z 257.383,A -85,B 0,C 180,E1 -11689.617,E2 -11689.617} C_VEL
LIN {X 0,Y 390.243,Z 257.371,A -85,B 0,C 180,E1 -11692.752,E2 -11692.752} C_VEL
LIN {X 0,Y 390.195,Z 257.377,A -85,B 0,C 180,E1 -11694.827,E2 -11694.827} C_VEL
LIN {X 0,Y 390.4,Z 257.356,A -85,B 0,C 180,E1 -11697.931,E2 -11697.931} C_VEL
LIN {X 0,Y 390.404,Z 257.353,A -85,B 0,C 180,E1 -11702.057,E2 -11702.057} C_VEL
LIN {X 0,Y 390.267,Z 257.368,A -85,B 0,C 180,E1 -11706.577,E2 -11706.577} C_VEL
LIN {X 0,Y 390.178,Z 257.385,A -85,B 0,C 180,E1 -11709.323,E2 -11709.323} C_VEL
LIN {X 0,Y 390.153,Z 257.382,A -85,B 0,C 180,E1 -11712.477,E2 -11712.477} C_VEL
LIN {X 0,Y 390.118,Z 257.389,A -85,B 0,C 180,E1 -11715.67,E2 -11715.67} C_VEL
LIN {X 0,Y 390.079,Z 257.396,A -85,B 0,C 180,E1 -11718.916,E2 -11718.916} C_VEL
LIN {X 0,Y 390.012,Z 257.4,A -85,B 0,C 180,E1 -11722.228,E2 -11722.228} C_VEL
LIN {X 0,Y 390.091,Z 257.39,A -85,B 0,C 180,E1 -11725.737,E2 -11725.737} C_VEL
LIN {X 0,Y 390.027,Z 257.401,A -85,B 0,C 180,E1 -11729.103,E2 -11729.103} C_VEL
LIN {X 0,Y 390.008,Z 257.407,A -85,B 0,C 180,E1 -11732.715,E2 -11732.715} C_VEL
LIN {X 0,Y 390.018,Z 257.399,A -85,B 0,C 180,E1 -11735.819,E2 -11735.819} C_VEL
LIN {X 0,Y 390.025,Z 257.399,A -85,B 0,C 180,E1 -11739.212,E2 -11739.212} C_VEL
LIN {X 0,Y 390.076,Z 257.398,A -85,B 0,C 180,E1 -11742.381,E2 -11742.381} C_VEL
LIN {X 0,Y 390.073,Z 257.392,A -85,B 0,C 180,E1 -11745.36,E2 -11745.36} C_VEL
LIN {X 0,Y 390.058,Z 257.4,A -85,B 0,C 180,E1 -11748.191,E2 -11748.191} C_VEL
LIN {X 0,Y 390.045,Z 257.396,A -85,B 0,C 180,E1 -11750.903,E2 -11750.903} C_VEL
LIN {X 0,Y 390.033,Z 257.398,A -85,B 0,C 180,E1 -11754.788,E2 -11754.788} C_VEL
LIN {X 0,Y 389.993,Z 257.404,A -85,B 0,C 180,E1 -11758.494,E2 -11758.494} C_VEL
LIN {X 0,Y 390.061,Z 257.398,A -85,B 0,C 180,E1 -11762.066,E2 -11762.066} C_VEL
LIN {X 0,Y 390.027,Z 257.402,A -85,B 0,C 180,E1 -11765.516,E2 -11765.516} C_VEL
LIN {X 0,Y 390.049,Z 257.395,A -85,B 0,C 180,E1 -11768.878,E2 -11768.878} C_VEL
LIN {X 0,Y 390.089,Z 257.395,A -85,B 0,C 180,E1 -11772.689,E2 -11772.689} C_VEL
LIN {X 0,Y 390.132,Z 257.39,A -85,B 0,C 180,E1 -11776.56,E2 -11776.56} C_VEL
LIN {X 0,Y 390.118,Z 257.391,A -85,B 0,C 180,E1 -11779.622,E2 -11779.622} C_VEL
LIN {X 0,Y 390.304,Z 257.455,A -85,B 0,C 180,E1 -11782.673,E2 -11782.673} C_VEL
LIN {X 0,Y 390.862,Z 259.444,A -85,B 0,C 180,E1 -11783.126,E2 -11783.126} C_VEL
LIN {X 0,Y 392.534,Z 261.797,A -85,B 0,C 180,E1 -11784.349,E2 -11784.349} C_VEL
LIN {X 0,Y 394.435,Z 263.063,A -85,B 0,C 180,E1 -11786.061,E2 -11786.061} C_VEL
LIN {X 0,Y 395.805,Z 263.405,A -85,B 0,C 180,E1 -11787.965,E2 -11787.965} C_VEL
LIN {X 0,Y 396.371,Z 263.477,A -85,B 0,C 180,E1 -11790,E2 -11790} C_VEL
LIN {X 0,Y 395.805,Z 263.405,A -85,B 0,C 180,E1 -11792.035,E2 -11792.035} C_VEL
LIN {X 0,Y 394.435,Z 263.056,A -85,B 0,C 180,E1 -11793.94,E2 -11793.94} C_VEL
LIN {X 0,Y 392.534,Z 261.797,A -85,B 0,C 180,E1 -11795.651,E2 -11795.651} C_VEL
LIN {X 0,Y 390.862,Z 259.444,A -85,B 0,C 180,E1 -11796.874,E2 -11796.874} C_VEL
LIN {X 0,Y 390.276,Z 257.373,A -85,B 0,C 180,E1 -11797.357,E2 -11797.357} C_VEL
